      movel(pose_trans(ref_frame,p[0.017484, 0.129054, -0.000125, -0.013708, 3.141563, 0.000000]),accel_mss,speed_ms,0,0.001)
      movel(pose_trans(ref_frame,p[0.017661, 0.129058, -0.000125, -0.013708, 3.141563, -0.000000]),accel_mss,speed_ms,0,0.001)
      movel(pose_trans(ref_frame,p[0.017837, 0.129065, -0.000125, -0.013708, 3.141563, -0.000000]),accel_mss,speed_ms,0,0.001)
      movel(pose_trans(ref_frame,p[0.017988, 0.129072, -0.000125, -0.013708, 3.141563, -0.000000]),accel_mss,speed_ms,0,0.001)
      movel(pose_trans(ref_frame,p[0.018138, 0.129080, -0.000125, -0.013708, 3.141563, 0.000000]),accel_mss,speed_ms,0,0.001)
      movel(pose_trans(ref_frame,p[0.018163, 0.129086, -0.000125, -0.013708, 3.141563, 0.000000]),accel_mss,speed_ms,0,0.001)
      movel(pose_trans(ref_frame,p[0.018184, 0.129101, -0.000125, -0.013708, 3.141563, -0.000000]),accel_mss,speed_ms,0,0.001)
      movel(pose_trans(ref_frame,p[0.018198, 0.129121, -0.000125, -0.013708, 3.141563, 0.000000]),accel_mss,speed_ms,0,0.001)
      movel(pose_trans(ref_frame,p[0.018205, 0.129145, -0.000125, -0.013708, 3.141563, 0.000000]),accel_mss,speed_ms,0,0.001)
      movel(pose_trans(ref_frame,p[0.018212, 0.129253, -0.000125, -0.013708, 3.141563, -0.000000]),accel_mss,speed_ms,0,0.001)
      movel(pose_trans(ref_frame,p[0.018218, 0.129360, -0.000125, -0.013708, 3.141563, -0.000000]),accel_mss,speed_ms,0,0.001)
      movel(pose_trans(ref_frame,p[0.018224, 0.129489, -0.000125, -0.013708, 3.141563, -0.000000]),accel_mss,speed_ms,0,0.001)
      movel(pose_trans(ref_frame,p[0.018228, 0.129617, -0.000125, -0.013708, 3.141563, 0.000000]),accel_mss,speed_ms,0,0.001)
      movel(pose_trans(ref_frame,p[0.018229, 0.129765, -0.000125, -0.013708, 3.141563, 0.000000]),accel_mss,speed_ms,0,0.001)
      movel(pose_trans(ref_frame,p[0.018229, 0.129912, -0.000125, -0.013708, 3.141563, -0.000000]),accel_mss,speed_ms,0,0.001)
      movel(pose_trans(ref_frame,p[0.018230, 0.130063, -0.000125, -0.013708, 3.141563, -0.000000]),accel_mss,speed_ms,0,0.001)
      movel(pose_trans(ref_frame,p[0.018236, 0.130213, -0.000125, -0.013708, 3.141563, -0.000000]),accel_mss,speed_ms,0,0.001)
      movel(pose_trans(ref_frame,p[0.018246, 0.130351, -0.000125, -0.013708, 3.141563, -0.000000]),accel_mss,speed_ms,0,0.001)
      movel(pose_trans(ref_frame,p[0.018262, 0.130488, -0.000125, -0.013708, 3.141563, -0.000000]),accel_mss,speed_ms,0,0.001)
      movel(pose_trans(ref_frame,p[0.018280, 0.130600, -0.000125, -0.013708, 3.141563, 0.000000]),accel_mss,speed_ms,0,0.001)
      movel(pose_trans(ref_frame,p[0.018302, 0.130711, -0.000125, -0.013708, 3.141563, -0.000000]),accel_mss,speed_ms,0,0.001)
      movel(pose_trans(ref_frame,p[0.018321, 0.130761, -0.000125, -0.013708, 3.141563, 0.000000]),accel_mss,speed_ms,0,0.001)
      movel(pose_trans(ref_frame,p[0.018353, 0.130804, -0.000125, -0.013708, 3.141563, 0.000000]),accel_mss,speed_ms,0,0.001)
      movel(pose_trans(ref_frame,p[0.018453, 0.130875, -0.000125, -0.013708, 3.141563, 0.000000]),accel_mss,speed_ms,0,0.001)
      movel(pose_trans(ref_frame,p[0.018570, 0.130910, -0.000125, -0.013708, 3.141563, -0.000000]),accel_mss,speed_ms,0,0.001)
      movel(pose_trans(ref_frame,p[0.018832, 0.130940, -0.000125, -0.013708, 3.141563, -0.000000]),accel_mss,speed_ms,0,0.001)
      movel(pose_trans(ref_frame,p[0.019095, 0.130958, -0.000125, -0.013708, 3.141563, -0.000000]),accel_mss,speed_ms,0,0.001)
      movel(pose_trans(ref_frame,p[0.019359, 0.130965, -0.000125, -0.013708, 3.141563, -0.000000]),accel_mss,speed_ms,0,0.001)
      movel(pose_trans(ref_frame,p[0.019623, 0.130962, -0.000125, -0.013708, 3.141563, 0.000000]),accel_mss,speed_ms,0,0.001)
      movel(pose_trans(ref_frame,p[0.019732, 0.130938, -0.000125, -0.013708, 3.141563, -0.000000]),accel_mss,speed_ms,0,0.001)
      movel(pose_trans(ref_frame,p[0.019825, 0.130874, -0.000125, -0.013708, 3.141563, -0.000000]),accel_mss,speed_ms,0,0.001)
      movel(pose_trans(ref_frame,p[0.019913, 0.130742, -0.000125, -0.013708, 3.141563, -0.000000]),accel_mss,speed_ms,0,0.001)
      movel(pose_trans(ref_frame,p[0.019945, 0.130587, -0.000125, -0.013708, 3.141563, -0.000000]),accel_mss,speed_ms,0,0.001)
      movel(pose_trans(ref_frame,p[0.019942, 0.129872, -0.000125, -0.013708, 3.141563, -0.000000]),accel_mss,speed_ms,0,0.001)
      movel(pose_trans(ref_frame,p[0.019933, 0.129158, -0.000125, -0.013708, 3.141563, -0.000000]),accel_mss,speed_ms,0,0.001)
      movel(pose_trans(ref_frame,p[0.019916, 0.128446, -0.000125, -0.013708, 3.141563, -0.000000]),accel_mss,speed_ms,0,0.001)
      movel(pose_trans(ref_frame,p[0.019891, 0.127733, -0.000125, -0.013708, 3.141563, -0.000000]),accel_mss,speed_ms,0,0.001)
      movel(pose_trans(ref_frame,p[0.019854, 0.127574, -0.000125, -0.013708, 3.141563, 0.000000]),accel_mss,speed_ms,0,0.001)
      movel(pose_trans(ref_frame,p[0.019761, 0.127438, -0.000125, -0.013708, 3.141563, -0.000000]),accel_mss,speed_ms,0,0.001)
      movel(pose_trans(ref_frame,p[0.019695, 0.127391, -0.000125, -0.013708, 3.141563, 0.000000]),accel_mss,speed_ms,0,0.001)
      movel(pose_trans(ref_frame,p[0.019616, 0.127368, -0.000125, -0.013708, 3.141563, -0.000000]),accel_mss,speed_ms,0,0.001)
      movel(pose_trans(ref_frame,p[0.019379, 0.127340, -0.000125, -0.013708, 3.141563, 0.000000]),accel_mss,speed_ms,0,0.001)
      movel(pose_trans(ref_frame,p[0.019142, 0.127318, -0.000125, -0.013708, 3.141563, -0.000000]),accel_mss,speed_ms,0,0.001)
      movel(pose_trans(ref_frame,p[0.018838, 0.127297, -0.000125, -0.013708, 3.141563, 0.000000]),accel_mss,speed_ms,0,0.001)
      movel(pose_trans(ref_frame,p[0.018535, 0.127285, -0.000125, -0.013708, 3.141563, 0.000000]),accel_mss,speed_ms,0,0.001)
      movel(pose_trans(ref_frame,p[0.018165, 0.127278, -0.000125, -0.013708, 3.141563, -0.000000]),accel_mss,speed_ms,0,0.001)
      movel(pose_trans(ref_frame,p[0.017795, 0.127276, -0.000125, -0.013708, 3.141563, -0.000000]),accel_mss,speed_ms,0,0.001)
      movel(pose_trans(ref_frame,p[0.015998, 0.127282, -0.000125, -0.013708, 3.141563, -0.000000]),accel_mss,speed_ms,0,0.001)
      movel(pose_trans(ref_frame,p[0.016051, 0.074830, -0.000125, -0.013708, 3.141563, 0.000000]),accel_mss,speed_ms,0,0.001)
      movel(pose_trans(ref_frame,p[0.016105, 0.022378, -0.000125, -0.013708, 3.141563, -0.000000]),accel_mss,speed_ms,0,0.001)
      movel(pose_trans(ref_frame,p[0.017978, 0.022373, -0.000125, -0.013708, 3.141563, -0.000000]),accel_mss,speed_ms,0,0.001)
      movel(pose_trans(ref_frame,p[0.018340, 0.022370, -0.000125, -0.013708, 3.141563, -0.000000]),accel_mss,speed_ms,0,0.001)
      movel(pose_trans(ref_frame,p[0.018702, 0.022365, -0.000125, -0.013708, 3.141563, -0.000000]),accel_mss,speed_ms,0,0.001)
      movel(pose_trans(ref_frame,p[0.019012, 0.022358, -0.000125, -0.013708, 3.141563, -0.000000]),accel_mss,speed_ms,0,0.001)
      movel(pose_trans(ref_frame,p[0.019323, 0.022347, -0.000125, -0.013708, 3.141563, -0.000000]),accel_mss,speed_ms,0,0.001)
      movel(pose_trans(ref_frame,p[0.019591, 0.022336, -0.000125, -0.013708, 3.141563, -0.000000]),accel_mss,speed_ms,0,0.001)
      movel(pose_trans(ref_frame,p[0.019858, 0.022323, -0.000125, -0.013708, 3.141563, 0.000000]),accel_mss,speed_ms,0,0.001)
      movel(pose_trans(ref_frame,p[0.019895, 0.022315, -0.000125, -0.013708, 3.141563, -0.000000]),accel_mss,speed_ms,0,0.001)
      movel(pose_trans(ref_frame,p[0.019925, 0.022294, -0.000125, -0.013708, 3.141563, -0.000000]),accel_mss,speed_ms,0,0.001)
      movel(pose_trans(ref_frame,p[0.019999, 0.022182, -0.000125, -0.013708, 3.141563, -0.000000]),accel_mss,speed_ms,0,0.001)
      movel(pose_trans(ref_frame,p[0.020024, 0.022051, -0.000125, -0.013708, 3.141563, 0.000000]),accel_mss,speed_ms,0,0.001)
      movel(pose_trans(ref_frame,p[0.020011, 0.021314, -0.000125, -0.013708, 3.141563, -0.000000]),accel_mss,speed_ms,0,0.001)
      movel(pose_trans(ref_frame,p[0.019994, 0.020578, -0.000125, -0.013708, 3.141563, -0.000000]),accel_mss,speed_ms,0,0.001)
      movel(pose_trans(ref_frame,p[0.019971, 0.019844, -0.000125, -0.013708, 3.141563, -0.000000]),accel_mss,speed_ms,0,0.001)
      movel(pose_trans(ref_frame,p[0.019943, 0.019110, -0.000125, -0.013708, 3.141563, -0.000000]),accel_mss,speed_ms,0,0.001)
      movel(pose_trans(ref_frame,p[0.019911, 0.018972, -0.000125, -0.013708, 3.141563, -0.000000]),accel_mss,speed_ms,0,0.001)
      movel(pose_trans(ref_frame,p[0.019832, 0.018856, -0.000125, -0.013708, 3.141563, -0.000000]),accel_mss,speed_ms,0,0.001)
      movel(pose_trans(ref_frame,p[0.019724, 0.018779, -0.000125, -0.013708, 3.141563, -0.000000]),accel_mss,speed_ms,0,0.001)
      movel(pose_trans(ref_frame,p[0.019598, 0.018740, -0.000125, -0.013708, 3.141563, 0.000000]),accel_mss,speed_ms,0,0.001)
      movel(pose_trans(ref_frame,p[0.019363, 0.018715, -0.000125, -0.013708, 3.141563, -0.000000]),accel_mss,speed_ms,0,0.001)
      movel(pose_trans(ref_frame,p[0.019127, 0.018706, -0.000125, -0.013708, 3.141563, 0.000000]),accel_mss,speed_ms,0,0.001)
      movel(pose_trans(ref_frame,p[0.018891, 0.018713, -0.000125, -0.013708, 3.141563, -0.000000]),accel_mss,speed_ms,0,0.001)
      movel(pose_trans(ref_frame,p[0.018657, 0.018735, -0.000125, -0.013708, 3.141563, 0.000000]),accel_mss,speed_ms,0,0.001)
      movel(pose_trans(ref_frame,p[0.018531, 0.018772, -0.000125, -0.013708, 3.141563, 0.000000]),accel_mss,speed_ms,0,0.001)
      movel(pose_trans(ref_frame,p[0.018424, 0.018848, -0.000125, -0.013708, 3.141563, -0.000000]),accel_mss,speed_ms,0,0.001)
      movel(pose_trans(ref_frame,p[0.018391, 0.018893, -0.000125, -0.013708, 3.141563, -0.000000]),accel_mss,speed_ms,0,0.001)
      movel(pose_trans(ref_frame,p[0.018370, 0.018945, -0.000125, -0.013708, 3.141563, -0.000000]),accel_mss,speed_ms,0,0.001)
      movel(pose_trans(ref_frame,p[0.018345, 0.019059, -0.000125, -0.013708, 3.141563, -0.000000]),accel_mss,speed_ms,0,0.001)
      movel(pose_trans(ref_frame,p[0.018324, 0.019174, -0.000125, -0.013708, 3.141563, -0.000000]),accel_mss,speed_ms,0,0.001)
      movel(pose_trans(ref_frame,p[0.018304, 0.019315, -0.000125, -0.013708, 3.141563, 0.000000]),accel_mss,speed_ms,0,0.001)
      movel(pose_trans(ref_frame,p[0.018290, 0.019456, -0.000125, -0.013708, 3.141563, -0.000000]),accel_mss,speed_ms,0,0.001)
      movel(pose_trans(ref_frame,p[0.018281, 0.019610, -0.000125, -0.013708, 3.141563, -0.000000]),accel_mss,speed_ms,0,0.001)
      movel(pose_trans(ref_frame,p[0.018276, 0.019764, -0.000125, -0.013708, 3.141563, -0.000000]),accel_mss,speed_ms,0,0.001)
      movel(pose_trans(ref_frame,p[0.018273, 0.019916, -0.000125, -0.013708, 3.141563, -0.000000]),accel_mss,speed_ms,0,0.001)
      movel(pose_trans(ref_frame,p[0.018267, 0.020067, -0.000125, -0.013708, 3.141563, 0.000000]),accel_mss,speed_ms,0,0.001)
      movel(pose_trans(ref_frame,p[0.018260, 0.020200, -0.000125, -0.013708, 3.141563, -0.000000]),accel_mss,speed_ms,0,0.001)
      movel(pose_trans(ref_frame,p[0.018249, 0.020333, -0.000125, -0.013708, 3.141563, -0.000000]),accel_mss,speed_ms,0,0.001)
      movel(pose_trans(ref_frame,p[0.018239, 0.020443, -0.000125, -0.013708, 3.141563, -0.000000]),accel_mss,speed_ms,0,0.001)
      movel(pose_trans(ref_frame,p[0.018227, 0.020553, -0.000125, -0.013708, 3.141563, -0.000000]),accel_mss,speed_ms,0,0.001)
      movel(pose_trans(ref_frame,p[0.018219, 0.020582, -0.000125, -0.013708, 3.141563, -0.000000]),accel_mss,speed_ms,0,0.001)
      movel(pose_trans(ref_frame,p[0.018201, 0.020606, -0.000125, -0.013708, 3.141563, -0.000000]),accel_mss,speed_ms,0,0.001)
      movel(pose_trans(ref_frame,p[0.018176, 0.020624, -0.000125, -0.013708, 3.141563, -0.000000]),accel_mss,speed_ms,0,0.001)
      movel(pose_trans(ref_frame,p[0.018146, 0.020632, -0.000125, -0.013708, 3.141563, -0.000000]),accel_mss,speed_ms,0,0.001)
      movel(pose_trans(ref_frame,p[0.018002, 0.020641, -0.000125, -0.013708, 3.141563, -0.000000]),accel_mss,speed_ms,0,0.001)
      movel(pose_trans(ref_frame,p[0.017857, 0.020649, -0.000125, -0.013708, 3.141563, -0.000000]),accel_mss,speed_ms,0,0.001)
      movel(pose_trans(ref_frame,p[0.017685, 0.020657, -0.000125, -0.013708, 3.141563, -0.000000]),accel_mss,speed_ms,0,0.001)
      movel(pose_trans(ref_frame,p[0.017514, 0.020662, -0.000125, -0.013708, 3.141563, -0.000000]),accel_mss,speed_ms,0,0.001)
      movel(pose_trans(ref_frame,p[0.017316, 0.020664, -0.000125, -0.013708, 3.141563, -0.000000]),accel_mss,speed_ms,0,0.001)
      movel(pose_trans(ref_frame,p[0.017118, 0.020664, -0.000125, -0.013708, 3.141563, -0.000000]),accel_mss,speed_ms,0,0.001)
      movel(pose_trans(ref_frame,p[0.016098, 0.020659, -0.000125, -0.013708, 3.141563, -0.000000]),accel_mss,speed_ms,0,0.001)
      movel(pose_trans(ref_frame,p[0.016098, 0.019605, -0.000125, -0.013708, 3.141563, -0.000000]),accel_mss,speed_ms,0,0.001)
      movel(pose_trans(ref_frame,p[0.016098, 0.018551, -0.000125, -0.013708, 3.141563, 0.000000]),accel_mss,speed_ms,0,0.001)
      movel(pose_trans(ref_frame,p[0.017009, 0.018525, -0.000125, -0.013708, 3.141563, -0.000000]),accel_mss,speed_ms,0,0.001)
      movel(pose_trans(ref_frame,p[0.017185, 0.018519, -0.000125, -0.013708, 3.141563, -0.000000]),accel_mss,speed_ms,0,0.001)
      movel(pose_trans(ref_frame,p[0.017362, 0.018512, -0.000125, -0.013708, 3.141563, -0.000000]),accel_mss,speed_ms,0,0.001)
      movel(pose_trans(ref_frame,p[0.017514, 0.018504, -0.000125, -0.013708, 3.141563, -0.000000]),accel_mss,speed_ms,0,0.001)
      movel(pose_trans(ref_frame,p[0.017666, 0.018493, -0.000125, -0.013708, 3.141563, -0.000000]),accel_mss,speed_ms,0,0.001)
      movel(pose_trans(ref_frame,p[0.017796, 0.018483, -0.000125, -0.013708, 3.141563, -0.000000]),accel_mss,speed_ms,0,0.001)
      movel(pose_trans(ref_frame,p[0.017925, 0.018472, -0.000125, -0.013708, 3.141563, 0.000000]),accel_mss,speed_ms,0,0.001)
      movel(pose_trans(ref_frame,p[0.017948, 0.018466, -0.000125, -0.013708, 3.141563, 0.000000]),accel_mss,speed_ms,0,0.001)
      movel(pose_trans(ref_frame,p[0.017968, 0.018452, -0.000125, -0.013708, 3.141563, 0.000000]),accel_mss,speed_ms,0,0.001)
      movel(pose_trans(ref_frame,p[0.018022, 0.018372, -0.000125, -0.013708, 3.141563, 0.000000]),accel_mss,speed_ms,0,0.001)
      movel(pose_trans(ref_frame,p[0.018043, 0.018278, -0.000125, -0.013708, 3.141563, -0.000000]),accel_mss,speed_ms,0,0.001)
      movel(pose_trans(ref_frame,p[0.018048, 0.017994, -0.000125, -0.013708, 3.141563, -0.000000]),accel_mss,speed_ms,0,0.001)
      movel(pose_trans(ref_frame,p[0.018046, 0.017710, -0.000125, -0.013708, 3.141563, -0.000000]),accel_mss,speed_ms,0,0.001)
      movel(pose_trans(ref_frame,p[0.018037, 0.017427, -0.000125, -0.013708, 3.141563, -0.000000]),accel_mss,speed_ms,0,0.001)
      movel(pose_trans(ref_frame,p[0.018022, 0.017143, -0.000125, -0.013708, 3.141563, -0.000000]),accel_mss,speed_ms,0,0.001)
      movel(pose_trans(ref_frame,p[0.017997, 0.017047, -0.000125, -0.013708, 3.141563, -0.000000]),accel_mss,speed_ms,0,0.001)
      movel(pose_trans(ref_frame,p[0.017940, 0.016965, -0.000125, -0.013708, 3.141563, -0.000000]),accel_mss,speed_ms,0,0.001)
      movel(pose_trans(ref_frame,p[0.017895, 0.016930, -0.000125, -0.013708, 3.141563, -0.000000]),accel_mss,speed_ms,0,0.001)
      movel(pose_trans(ref_frame,p[0.017843, 0.016910, -0.000125, -0.013708, 3.141563, -0.000000]),accel_mss,speed_ms,0,0.001)
      movel(pose_trans(ref_frame,p[0.017730, 0.016885, -0.000125, -0.013708, 3.141563, -0.000000]),accel_mss,speed_ms,0,0.001)
      movel(pose_trans(ref_frame,p[0.017617, 0.016865, -0.000125, -0.013708, 3.141563, -0.000000]),accel_mss,speed_ms,0,0.001)
      movel(pose_trans(ref_frame,p[0.017478, 0.016846, -0.000125, -0.013708, 3.141563, -0.000000]),accel_mss,speed_ms,0,0.001)
      movel(pose_trans(ref_frame,p[0.017339, 0.016833, -0.000125, -0.013708, 3.141563, -0.000000]),accel_mss,speed_ms,0,0.001)
      movel(pose_trans(ref_frame,p[0.017188, 0.016825, -0.000125, -0.013708, 3.141563, -0.000000]),accel_mss,speed_ms,0,0.001)
      movel(pose_trans(ref_frame,p[0.017036, 0.016823, -0.000125, -0.013708, 3.141563, 0.000000]),accel_mss,speed_ms,0,0.001)
      movel(pose_trans(ref_frame,p[0.016887, 0.016821, -0.000125, -0.013708, 3.141563, -0.000000]),accel_mss,speed_ms,0,0.001)
      movel(pose_trans(ref_frame,p[0.016737, 0.016816, -0.000125, -0.013708, 3.141563, -0.000000]),accel_mss,speed_ms,0,0.001)
      movel(pose_trans(ref_frame,p[0.016604, 0.016808, -0.000125, -0.013708, 3.141563, -0.000000]),accel_mss,speed_ms,0,0.001)
      movel(pose_trans(ref_frame,p[0.016470, 0.016796, -0.000125, -0.013708, 3.141563, -0.000000]),accel_mss,speed_ms,0,0.001)
      movel(pose_trans(ref_frame,p[0.016361, 0.016784, -0.000125, -0.013708, 3.141563, -0.000000]),accel_mss,speed_ms,0,0.001)
      movel(pose_trans(ref_frame,p[0.016252, 0.016769, -0.000125, -0.013708, 3.141563, -0.000000]),accel_mss,speed_ms,0,0.001)
      movel(pose_trans(ref_frame,p[0.016214, 0.016758, -0.000125, -0.013708, 3.141563, -0.000000]),accel_mss,speed_ms,0,0.001)
      movel(pose_trans(ref_frame,p[0.016182, 0.016736, -0.000125, -0.013708, 3.141563, -0.000000]),accel_mss,speed_ms,0,0.001)
      movel(pose_trans(ref_frame,p[0.016158, 0.016703, -0.000125, -0.013708, 3.141563, -0.000000]),accel_mss,speed_ms,0,0.001)
      movel(pose_trans(ref_frame,p[0.016146, 0.016664, -0.000125, -0.013708, 3.141563, -0.000000]),accel_mss,speed_ms,0,0.001)
      movel(pose_trans(ref_frame,p[0.016132, 0.016520, -0.000125, -0.013708, 3.141563, -0.000000]),accel_mss,speed_ms,0,0.001)
      movel(pose_trans(ref_frame,p[0.016119, 0.016377, -0.000125, -0.013708, 3.141563, -0.000000]),accel_mss,speed_ms,0,0.001)
      movel(pose_trans(ref_frame,p[0.016108, 0.016203, -0.000125, -0.013708, 3.141563, 0.000000]),accel_mss,speed_ms,0,0.001)
      movel(pose_trans(ref_frame,p[0.016101, 0.016029, -0.000125, -0.013708, 3.141563, 0.000000]),accel_mss,speed_ms,0,0.001)
      movel(pose_trans(ref_frame,p[0.016097, 0.015831, -0.000125, -0.013708, 3.141563, -0.000000]),accel_mss,speed_ms,0,0.001)
      movel(pose_trans(ref_frame,p[0.016097, 0.015633, -0.000125, -0.013708, 3.141563, -0.000000]),accel_mss,speed_ms,0,0.001)
      movel(pose_trans(ref_frame,p[0.016102, 0.014616, -0.000125, -0.013708, 3.141563, -0.000000]),accel_mss,speed_ms,0,0.001)
      movel(pose_trans(ref_frame,p[0.016912, 0.014609, -0.000125, -0.013708, 3.141563, -0.000000]),accel_mss,speed_ms,0,0.001)
      movel(pose_trans(ref_frame,p[0.017074, 0.014605, -0.000125, -0.013708, 3.141563, -0.000000]),accel_mss,speed_ms,0,0.001)
      movel(pose_trans(ref_frame,p[0.017235, 0.014595, -0.000125, -0.013708, 3.141563, -0.000000]),accel_mss,speed_ms,0,0.001)
      movel(pose_trans(ref_frame,p[0.017384, 0.014579, -0.000125, -0.013708, 3.141563, -0.000000]),accel_mss,speed_ms,0,0.001)
      movel(pose_trans(ref_frame,p[0.017533, 0.014557, -0.000125, -0.013708, 3.141563, -0.000000]),accel_mss,speed_ms,0,0.001)
      movel(pose_trans(ref_frame,p[0.017655, 0.014533, -0.000125, -0.013708, 3.141563, -0.000000]),accel_mss,speed_ms,0,0.001)
      movel(pose_trans(ref_frame,p[0.017776, 0.014503, -0.000125, -0.013708, 3.141563, -0.000000]),accel_mss,speed_ms,0,0.001)
      movel(pose_trans(ref_frame,p[0.017836, 0.014478, -0.000125, -0.013708, 3.141563, -0.000000]),accel_mss,speed_ms,0,0.001)
      movel(pose_trans(ref_frame,p[0.017888, 0.014438, -0.000125, -0.013708, 3.141563, -0.000000]),accel_mss,speed_ms,0,0.001)
      movel(pose_trans(ref_frame,p[0.017927, 0.014387, -0.000125, -0.013708, 3.141563, -0.000000]),accel_mss,speed_ms,0,0.001)
      movel(pose_trans(ref_frame,p[0.017952, 0.014327, -0.000125, -0.013708, 3.141563, -0.000000]),accel_mss,speed_ms,0,0.001)
      movel(pose_trans(ref_frame,p[0.017982, 0.014206, -0.000125, -0.013708, 3.141563, -0.000000]),accel_mss,speed_ms,0,0.001)
      movel(pose_trans(ref_frame,p[0.018006, 0.014084, -0.000125, -0.013708, 3.141563, 0.000000]),accel_mss,speed_ms,0,0.001)
      movel(pose_trans(ref_frame,p[0.018028, 0.013935, -0.000125, -0.013708, 3.141563, 0.000000]),accel_mss,speed_ms,0,0.001)
      movel(pose_trans(ref_frame,p[0.018044, 0.013786, -0.000125, -0.013708, 3.141563, -0.000000]),accel_mss,speed_ms,0,0.001)
      movel(pose_trans(ref_frame,p[0.018054, 0.013625, -0.000125, -0.013708, 3.141563, -0.000000]),accel_mss,speed_ms,0,0.001)
      movel(pose_trans(ref_frame,p[0.018058, 0.013463, -0.000125, -0.013708, 3.141563, -0.000000]),accel_mss,speed_ms,0,0.001)
      movel(pose_trans(ref_frame,p[0.018065, 0.012653, -0.000125, -0.013708, 3.141563, -0.000000]),accel_mss,speed_ms,0,0.001)
      movel(pose_trans(ref_frame,p[0.019082, 0.012648, -0.000125, -0.013708, 3.141563, -0.000000]),accel_mss,speed_ms,0,0.001)
      movel(pose_trans(ref_frame,p[0.019281, 0.012648, -0.000125, -0.013708, 3.141563, 0.000000]),accel_mss,speed_ms,0,0.001)
      movel(pose_trans(ref_frame,p[0.019479, 0.012653, -0.000125, -0.013708, 3.141563, -0.000000]),accel_mss,speed_ms,0,0.001)
      movel(pose_trans(ref_frame,p[0.019654, 0.012660, -0.000125, -0.013708, 3.141563, -0.000000]),accel_mss,speed_ms,0,0.001)
      movel(pose_trans(ref_frame,p[0.019830, 0.012673, -0.000125, -0.013708, 3.141563, -0.000000]),accel_mss,speed_ms,0,0.001)
      movel(pose_trans(ref_frame,p[0.019974, 0.012686, -0.000125, -0.013708, 3.141563, -0.000000]),accel_mss,speed_ms,0,0.001)
      movel(pose_trans(ref_frame,p[0.020118, 0.012702, -0.000125, -0.013708, 3.141563, -0.000000]),accel_mss,speed_ms,0,0.001)
      movel(pose_trans(ref_frame,p[0.020161, 0.012715, -0.000125, -0.013708, 3.141563, -0.000000]),accel_mss,speed_ms,0,0.001)
      movel(pose_trans(ref_frame,p[0.020198, 0.012741, -0.000125, -0.013708, 3.141563, -0.000000]),accel_mss,speed_ms,0,0.001)
      movel(pose_trans(ref_frame,p[0.020223, 0.012775, -0.000125, -0.013708, 3.141563, -0.000000]),accel_mss,speed_ms,0,0.001)
      movel(pose_trans(ref_frame,p[0.020235, 0.012815, -0.000125, -0.013708, 3.141563, -0.000000]),accel_mss,speed_ms,0,0.001)
      movel(pose_trans(ref_frame,p[0.020248, 0.012921, -0.000125, -0.013708, 3.141563, -0.000000]),accel_mss,speed_ms,0,0.001)
      movel(pose_trans(ref_frame,p[0.020259, 0.013027, -0.000125, -0.013708, 3.141563, -0.000000]),accel_mss,speed_ms,0,0.001)
      movel(pose_trans(ref_frame,p[0.020267, 0.013157, -0.000125, -0.013708, 3.141563, -0.000000]),accel_mss,speed_ms,0,0.001)
      movel(pose_trans(ref_frame,p[0.020271, 0.013287, -0.000125, -0.013708, 3.141563, -0.000000]),accel_mss,speed_ms,0,0.001)
      movel(pose_trans(ref_frame,p[0.020270, 0.013432, -0.000125, -0.013708, 3.141563, 0.000000]),accel_mss,speed_ms,0,0.001)
      movel(pose_trans(ref_frame,p[0.020266, 0.013577, -0.000125, -0.013708, 3.141563, 0.000000]),accel_mss,speed_ms,0,0.001)
      movel(pose_trans(ref_frame,p[0.020263, 0.013723, -0.000125, -0.013708, 3.141563, -0.000000]),accel_mss,speed_ms,0,0.001)
      movel(pose_trans(ref_frame,p[0.020266, 0.013870, -0.000125, -0.013708, 3.141563, -0.000000]),accel_mss,speed_ms,0,0.001)
      movel(pose_trans(ref_frame,p[0.020275, 0.014006, -0.000125, -0.013708, 3.141563, -0.000000]),accel_mss,speed_ms,0,0.001)
      movel(pose_trans(ref_frame,p[0.020290, 0.014142, -0.000125, -0.013708, 3.141563, 0.000000]),accel_mss,speed_ms,0,0.001)
      movel(pose_trans(ref_frame,p[0.020308, 0.014253, -0.000125, -0.013708, 3.141563, -0.000000]),accel_mss,speed_ms,0,0.001)
      movel(pose_trans(ref_frame,p[0.020331, 0.014364, -0.000125, -0.013708, 3.141563, -0.000000]),accel_mss,speed_ms,0,0.001)
      movel(pose_trans(ref_frame,p[0.020353, 0.014419, -0.000125, -0.013708, 3.141563, -0.000000]),accel_mss,speed_ms,0,0.001)
      movel(pose_trans(ref_frame,p[0.020389, 0.014466, -0.000125, -0.013708, 3.141563, -0.000000]),accel_mss,speed_ms,0,0.001)
      movel(pose_trans(ref_frame,p[0.020498, 0.014544, -0.000125, -0.013708, 3.141563, -0.000000]),accel_mss,speed_ms,0,0.001)
      movel(pose_trans(ref_frame,p[0.020626, 0.014582, -0.000125, -0.013708, 3.141563, -0.000000]),accel_mss,speed_ms,0,0.001)
      movel(pose_trans(ref_frame,p[0.020861, 0.014602, -0.000125, -0.013708, 3.141563, -0.000000]),accel_mss,speed_ms,0,0.001)
      movel(pose_trans(ref_frame,p[0.021097, 0.014605, -0.000125, -0.013708, 3.141563, -0.000000]),accel_mss,speed_ms,0,0.001)
      movel(pose_trans(ref_frame,p[0.021333, 0.014592, -0.000125, -0.013708, 3.141563, -0.000000]),accel_mss,speed_ms,0,0.001)
      movel(pose_trans(ref_frame,p[0.021568, 0.014562, -0.000125, -0.013708, 3.141563, -0.000000]),accel_mss,speed_ms,0,0.001)
      movel(pose_trans(ref_frame,p[0.021700, 0.014519, -0.000125, -0.013708, 3.141563, -0.000000]),accel_mss,speed_ms,0,0.001)
      movel(pose_trans(ref_frame,p[0.021812, 0.014437, -0.000125, -0.013708, 3.141563, -0.000000]),accel_mss,speed_ms,0,0.001)
      movel(pose_trans(ref_frame,p[0.021851, 0.014386, -0.000125, -0.013708, 3.141563, -0.000000]),accel_mss,speed_ms,0,0.001)
      movel(pose_trans(ref_frame,p[0.021876, 0.014326, -0.000125, -0.013708, 3.141563, -0.000000]),accel_mss,speed_ms,0,0.001)
      movel(pose_trans(ref_frame,p[0.021905, 0.014205, -0.000125, -0.013708, 3.141563, 0.000000]),accel_mss,speed_ms,0,0.001)
      movel(pose_trans(ref_frame,p[0.021929, 0.014083, -0.000125, -0.013708, 3.141563, -0.000000]),accel_mss,speed_ms,0,0.001)
      movel(pose_trans(ref_frame,p[0.021951, 0.013934, -0.000125, -0.013708, 3.141563, -0.000000]),accel_mss,speed_ms,0,0.001)
      movel(pose_trans(ref_frame,p[0.021967, 0.013784, -0.000125, -0.013708, 3.141563, -0.000000]),accel_mss,speed_ms,0,0.001)
      movel(pose_trans(ref_frame,p[0.021977, 0.013623, -0.000125, -0.013708, 3.141563, -0.000000]),accel_mss,speed_ms,0,0.001)
      movel(pose_trans(ref_frame,p[0.021982, 0.013462, -0.000125, -0.013708, 3.141563, 0.000000]),accel_mss,speed_ms,0,0.001)
      movel(pose_trans(ref_frame,p[0.021988, 0.012649, -0.000125, -0.013708, 3.141563, -0.000000]),accel_mss,speed_ms,0,0.001)
      movel(pose_trans(ref_frame,p[0.023048, 0.012649, -0.000125, -0.013708, 3.141563, -0.000000]),accel_mss,speed_ms,0,0.001)
      movel(pose_trans(ref_frame,p[0.024108, 0.012649, -0.000125, -0.013708, 3.141563, -0.000000]),accel_mss,speed_ms,0,0.001)
      movel(pose_trans(ref_frame,p[0.024113, 0.013669, -0.000125, -0.013708, 3.141563, -0.000000]),accel_mss,speed_ms,0,0.001)
      movel(pose_trans(ref_frame,p[0.024113, 0.013866, -0.000125, -0.013708, 3.141563, -0.000000]),accel_mss,speed_ms,0,0.001)
      movel(pose_trans(ref_frame,p[0.024112, 0.014063, -0.000125, -0.013708, 3.141563, -0.000000]),accel_mss,speed_ms,0,0.001)
      movel(pose_trans(ref_frame,p[0.024109, 0.014233, -0.000125, -0.013708, 3.141563, 0.000000]),accel_mss,speed_ms,0,0.001)
      movel(pose_trans(ref_frame,p[0.024103, 0.014403, -0.000125, -0.013708, 3.141563, -0.000000]),accel_mss,speed_ms,0,0.001)
      movel(pose_trans(ref_frame,p[0.024098, 0.014548, -0.000125, -0.013708, 3.141563, -0.000000]),accel_mss,speed_ms,0,0.001)
      movel(pose_trans(ref_frame,p[0.024091, 0.014693, -0.000125, -0.013708, 3.141563, -0.000000]),accel_mss,speed_ms,0,0.001)
      movel(pose_trans(ref_frame,p[0.024086, 0.014716, -0.000125, -0.013708, 3.141563, -0.000000]),accel_mss,speed_ms,0,0.001)
      movel(pose_trans(ref_frame,p[0.024073, 0.014735, -0.000125, -0.013708, 3.141563, -0.000000]),accel_mss,speed_ms,0,0.001)
      movel(pose_trans(ref_frame,p[0.024054, 0.014748, -0.000125, -0.013708, 3.141563, -0.000000]),accel_mss,speed_ms,0,0.001)
      movel(pose_trans(ref_frame,p[0.024032, 0.014755, -0.000125, -0.013708, 3.141563, -0.000000]),accel_mss,speed_ms,0,0.001)
      movel(pose_trans(ref_frame,p[0.023918, 0.014768, -0.000125, -0.013708, 3.141563, -0.000000]),accel_mss,speed_ms,0,0.001)
      movel(pose_trans(ref_frame,p[0.023803, 0.014780, -0.000125, -0.013708, 3.141563, -0.000000]),accel_mss,speed_ms,0,0.001)
      movel(pose_trans(ref_frame,p[0.023667, 0.014793, -0.000125, -0.013708, 3.141563, -0.000000]),accel_mss,speed_ms,0,0.001)
      movel(pose_trans(ref_frame,p[0.023532, 0.014804, -0.000125, -0.013708, 3.141563, 0.000000]),accel_mss,speed_ms,0,0.001)
      movel(pose_trans(ref_frame,p[0.023375, 0.014815, -0.000125, -0.013708, 3.141563, 0.000000]),accel_mss,speed_ms,0,0.001)
      movel(pose_trans(ref_frame,p[0.023218, 0.014824, -0.000125, -0.013708, 3.141563, -0.000000]),accel_mss,speed_ms,0,0.001)
      movel(pose_trans(ref_frame,p[0.023059, 0.014835, -0.000125, -0.013708, 3.141563, -0.000000]),accel_mss,speed_ms,0,0.001)
      movel(pose_trans(ref_frame,p[0.022899, 0.014850, -0.000125, -0.013708, 3.141563, 0.000000]),accel_mss,speed_ms,0,0.001)
      movel(pose_trans(ref_frame,p[0.022753, 0.014869, -0.000125, -0.013708, 3.141563, -0.000000]),accel_mss,speed_ms,0,0.001)
      movel(pose_trans(ref_frame,p[0.022608, 0.014893, -0.000125, -0.013708, 3.141563, -0.000000]),accel_mss,speed_ms,0,0.001)
      movel(pose_trans(ref_frame,p[0.022490, 0.014917, -0.000125, -0.013708, 3.141563, -0.000000]),accel_mss,speed_ms,0,0.001)
      movel(pose_trans(ref_frame,p[0.022372, 0.014945, -0.000125, -0.013708, 3.141563, -0.000000]),accel_mss,speed_ms,0,0.001)
      movel(pose_trans(ref_frame,p[0.022321, 0.014966, -0.000125, -0.013708, 3.141563, -0.000000]),accel_mss,speed_ms,0,0.001)
      movel(pose_trans(ref_frame,p[0.022276, 0.014999, -0.000125, -0.013708, 3.141563, -0.000000]),accel_mss,speed_ms,0,0.001)
      movel(pose_trans(ref_frame,p[0.022205, 0.015098, -0.000125, -0.013708, 3.141563, 0.000000]),accel_mss,speed_ms,0,0.001)
      movel(pose_trans(ref_frame,p[0.022173, 0.015216, -0.000125, -0.013708, 3.141563, -0.000000]),accel_mss,speed_ms,0,0.001)
      movel(pose_trans(ref_frame,p[0.022157, 0.015451, -0.000125, -0.013708, 3.141563, -0.000000]),accel_mss,speed_ms,0,0.001)
      movel(pose_trans(ref_frame,p[0.022155, 0.015687, -0.000125, -0.013708, 3.141563, -0.000000]),accel_mss,speed_ms,0,0.001)
      movel(pose_trans(ref_frame,p[0.022167, 0.015923, -0.000125, -0.013708, 3.141563, -0.000000]),accel_mss,speed_ms,0,0.001)
      movel(pose_trans(ref_frame,p[0.022193, 0.016158, -0.000125, -0.013708, 3.141563, 0.000000]),accel_mss,speed_ms,0,0.001)
      movel(pose_trans(ref_frame,p[0.022232, 0.016280, -0.000125, -0.013708, 3.141563, -0.000000]),accel_mss,speed_ms,0,0.001)
      movel(pose_trans(ref_frame,p[0.022306, 0.016384, -0.000125, -0.013708, 3.141563, -0.000000]),accel_mss,speed_ms,0,0.001)
      movel(pose_trans(ref_frame,p[0.022407, 0.016453, -0.000125, -0.013708, 3.141563, -0.000000]),accel_mss,speed_ms,0,0.001)
      movel(pose_trans(ref_frame,p[0.022526, 0.016479, -0.000125, -0.013708, 3.141563, -0.000000]),accel_mss,speed_ms,0,0.001)
      movel(pose_trans(ref_frame,p[0.023281, 0.016501, -0.000125, -0.013708, 3.141563, -0.000000]),accel_mss,speed_ms,0,0.001)
      movel(pose_trans(ref_frame,p[0.024036, 0.016519, -0.000125, -0.013708, 3.141563, -0.000000]),accel_mss,speed_ms,0,0.001)
      movel(pose_trans(ref_frame,p[0.024793, 0.016533, -0.000125, -0.013708, 3.141563, -0.000000]),accel_mss,speed_ms,0,0.001)
      movel(pose_trans(ref_frame,p[0.025550, 0.016544, -0.000125, -0.013708, 3.141563, 0.000000]),accel_mss,speed_ms,0,0.001)
      movel(pose_trans(ref_frame,p[0.025665, 0.016522, -0.000125, -0.013708, 3.141563, 0.000000]),accel_mss,speed_ms,0,0.001)
      movel(pose_trans(ref_frame,p[0.025762, 0.016457, -0.000125, -0.013708, 3.141563, -0.000000]),accel_mss,speed_ms,0,0.001)
      movel(pose_trans(ref_frame,p[0.025778, 0.016434, -0.000125, -0.013708, 3.141563, -0.000000]),accel_mss,speed_ms,0,0.001)
      movel(pose_trans(ref_frame,p[0.025784, 0.016406, -0.000125, -0.013708, 3.141563, -0.000000]),accel_mss,speed_ms,0,0.001)
      movel(pose_trans(ref_frame,p[0.025793, 0.016137, -0.000125, -0.013708, 3.141563, -0.000000]),accel_mss,speed_ms,0,0.001)
      movel(pose_trans(ref_frame,p[0.025801, 0.015868, -0.000125, -0.013708, 3.141563, -0.000000]),accel_mss,speed_ms,0,0.001)
      movel(pose_trans(ref_frame,p[0.025809, 0.015559, -0.000125, -0.013708, 3.141563, 0.000000]),accel_mss,speed_ms,0,0.001)
      movel(pose_trans(ref_frame,p[0.025814, 0.015250, -0.000125, -0.013708, 3.141563, -0.000000]),accel_mss,speed_ms,0,0.001)
      movel(pose_trans(ref_frame,p[0.025818, 0.014889, -0.000125, -0.013708, 3.141563, 0.000000]),accel_mss,speed_ms,0,0.001)
      movel(pose_trans(ref_frame,p[0.025820, 0.014527, -0.000125, -0.013708, 3.141563, -0.000000]),accel_mss,speed_ms,0,0.001)
      movel(pose_trans(ref_frame,p[0.025823, 0.012652, -0.000125, -0.013708, 3.141563, 0.000000]),accel_mss,speed_ms,0,0.001)
      movel(pose_trans(ref_frame,p[0.078266, 0.012593, -0.000125, -0.013708, 3.141563, -0.000000]),accel_mss,speed_ms,0,0.001)
      movel(pose_trans(ref_frame,p[0.130708, 0.012535, -0.000125, -0.013708, 3.141563, 0.000000]),accel_mss,speed_ms,0,0.001)
      movel(pose_trans(ref_frame,p[0.130721, 0.014348, -0.000125, -0.013708, 3.141563, -0.000000]),accel_mss,speed_ms,0,0.001)
      movel(pose_trans(ref_frame,p[0.130726, 0.014701, -0.000125, -0.013708, 3.141563, -0.000000]),accel_mss,speed_ms,0,0.001)
      movel(pose_trans(ref_frame,p[0.130736, 0.015053, -0.000125, -0.013708, 3.141563, -0.000000]),accel_mss,speed_ms,0,0.001)
      movel(pose_trans(ref_frame,p[0.130750, 0.015361, -0.000125, -0.013708, 3.141563, -0.000000]),accel_mss,speed_ms,0,0.001)
      movel(pose_trans(ref_frame,p[0.130771, 0.015669, -0.000125, -0.013708, 3.141563, -0.000000]),accel_mss,speed_ms,0,0.001)
      movel(pose_trans(ref_frame,p[0.130792, 0.015926, -0.000125, -0.013708, 3.141563, 0.000000]),accel_mss,speed_ms,0,0.001)
      movel(pose_trans(ref_frame,p[0.130816, 0.016182, -0.000125, -0.013708, 3.141563, -0.000000]),accel_mss,speed_ms,0,0.001)
      movel(pose_trans(ref_frame,p[0.130834, 0.016245, -0.000125, -0.013708, 3.141563, -0.000000]),accel_mss,speed_ms,0,0.001)
      movel(pose_trans(ref_frame,p[0.130871, 0.016298, -0.000125, -0.013708, 3.141563, -0.000000]),accel_mss,speed_ms,0,0.001)
      movel(pose_trans(ref_frame,p[0.130924, 0.016335, -0.000125, -0.013708, 3.141563, -0.000000]),accel_mss,speed_ms,0,0.001)
      movel(pose_trans(ref_frame,p[0.130985, 0.016353, -0.000125, -0.013708, 3.141563, 0.000000]),accel_mss,speed_ms,0,0.001)
      movel(pose_trans(ref_frame,p[0.131215, 0.016377, -0.000125, -0.013708, 3.141563, -0.000000]),accel_mss,speed_ms,0,0.001)
      movel(pose_trans(ref_frame,p[0.131445, 0.016399, -0.000125, -0.013708, 3.141563, 0.000000]),accel_mss,speed_ms,0,0.001)
      movel(pose_trans(ref_frame,p[0.131723, 0.016419, -0.000125, -0.013708, 3.141563, 0.000000]),accel_mss,speed_ms,0,0.001)
      movel(pose_trans(ref_frame,p[0.132001, 0.016434, -0.000125, -0.013708, 3.141563, 0.000000]),accel_mss,speed_ms,0,0.001)
      movel(pose_trans(ref_frame,p[0.132317, 0.016444, -0.000125, -0.013708, 3.141563, 0.000000]),accel_mss,speed_ms,0,0.001)
      movel(pose_trans(ref_frame,p[0.132633, 0.016449, -0.000125, -0.013708, 3.141563, -0.000000]),accel_mss,speed_ms,0,0.001)
      movel(pose_trans(ref_frame,p[0.133218, 0.016450, -0.000125, -0.013708, 3.141563, -0.000000]),accel_mss,speed_ms,0,0.001)
      movel(pose_trans(ref_frame,p[0.133803, 0.016442, -0.000125, -0.013708, 3.141563, -0.000000]),accel_mss,speed_ms,0,0.001)
      movel(pose_trans(ref_frame,p[0.134003, 0.016415, -0.000125, -0.013708, 3.141563, 0.000000]),accel_mss,speed_ms,0,0.001)
      movel(pose_trans(ref_frame,p[0.134192, 0.016343, -0.000125, -0.013708, 3.141563, -0.000000]),accel_mss,speed_ms,0,0.001)
      movel(pose_trans(ref_frame,p[0.134310, 0.016242, -0.000125, -0.013708, 3.141563, 0.000000]),accel_mss,speed_ms,0,0.001)
      movel(pose_trans(ref_frame,p[0.134370, 0.016099, -0.000125, -0.013708, 3.141563, -0.000000]),accel_mss,speed_ms,0,0.001)
      movel(pose_trans(ref_frame,p[0.134407, 0.015813, -0.000125, -0.013708, 3.141563, -0.000000]),accel_mss,speed_ms,0,0.001)
      movel(pose_trans(ref_frame,p[0.134420, 0.015525, -0.000125, -0.013708, 3.141563, -0.000000]),accel_mss,speed_ms,0,0.001)
      movel(pose_trans(ref_frame,p[0.134410, 0.015304, -0.000125, -0.013708, 3.141563, -0.000000]),accel_mss,speed_ms,0,0.001)
      movel(pose_trans(ref_frame,p[0.134382, 0.015084, -0.000125, -0.013708, 3.141563, -0.000000]),accel_mss,speed_ms,0,0.001)
      movel(pose_trans(ref_frame,p[0.134337, 0.014963, -0.000125, -0.013708, 3.141563, -0.000000]),accel_mss,speed_ms,0,0.001)
      movel(pose_trans(ref_frame,p[0.134251, 0.014867, -0.000125, -0.013708, 3.141563, -0.000000]),accel_mss,speed_ms,0,0.001)
      movel(pose_trans(ref_frame,p[0.134123, 0.014796, -0.000125, -0.013708, 3.141563, -0.000000]),accel_mss,speed_ms,0,0.001)
      movel(pose_trans(ref_frame,p[0.133980, 0.014763, -0.000125, -0.013708, 3.141563, 0.000000]),accel_mss,speed_ms,0,0.001)
      movel(pose_trans(ref_frame,p[0.133681, 0.014744, -0.000125, -0.013708, 3.141563, -0.000000]),accel_mss,speed_ms,0,0.001)
      movel(pose_trans(ref_frame,p[0.133382, 0.014737, -0.000125, -0.013708, 3.141563, -0.000000]),accel_mss,speed_ms,0,0.001)
      movel(pose_trans(ref_frame,p[0.132513, 0.014735, -0.000125, -0.013708, 3.141563, -0.000000]),accel_mss,speed_ms,0,0.001)
      movel(pose_trans(ref_frame,p[0.132508, 0.013651, -0.000125, -0.013708, 3.141563, 0.000000]),accel_mss,speed_ms,0,0.001)
      movel(pose_trans(ref_frame,p[0.132503, 0.012567, -0.000125, -0.013708, 3.141563, -0.000000]),accel_mss,speed_ms,0,0.001)
      movel(pose_trans(ref_frame,p[0.133569, 0.012562, -0.000125, -0.013708, 3.141563, -0.000000]),accel_mss,speed_ms,0,0.001)
      movel(pose_trans(ref_frame,p[0.134635, 0.012557, -0.000125, -0.013708, 3.141563, -0.000000]),accel_mss,speed_ms,0,0.001)
      movel(pose_trans(ref_frame,p[0.134640, 0.013415, -0.000125, -0.013708, 3.141563, -0.000000]),accel_mss,speed_ms,0,0.001)
      movel(pose_trans(ref_frame,p[0.134644, 0.013585, -0.000125, -0.013708, 3.141563, 0.000000]),accel_mss,speed_ms,0,0.001)
      movel(pose_trans(ref_frame,p[0.134652, 0.013754, -0.000125, -0.013708, 3.141563, -0.000000]),accel_mss,speed_ms,0,0.001)
      movel(pose_trans(ref_frame,p[0.134664, 0.013907, -0.000125, -0.013708, 3.141563, 0.000000]),accel_mss,speed_ms,0,0.001)
      movel(pose_trans(ref_frame,p[0.134682, 0.014060, -0.000125, -0.013708, 3.141563, -0.000000]),accel_mss,speed_ms,0,0.001)
      movel(pose_trans(ref_frame,p[0.134702, 0.014184, -0.000125, -0.013708, 3.141563, -0.000000]),accel_mss,speed_ms,0,0.001)
      movel(pose_trans(ref_frame,p[0.134725, 0.014308, -0.000125, -0.013708, 3.141563, -0.000000]),accel_mss,speed_ms,0,0.001)
      movel(pose_trans(ref_frame,p[0.134743, 0.014360, -0.000125, -0.013708, 3.141563, -0.000000]),accel_mss,speed_ms,0,0.001)
      movel(pose_trans(ref_frame,p[0.134776, 0.014404, -0.000125, -0.013708, 3.141563, -0.000000]),accel_mss,speed_ms,0,0.001)
      movel(pose_trans(ref_frame,p[0.134843, 0.014453, -0.000125, -0.013708, 3.141563, -0.000000]),accel_mss,speed_ms,0,0.001)
      movel(pose_trans(ref_frame,p[0.134922, 0.014478, -0.000125, -0.013708, 3.141563, -0.000000]),accel_mss,speed_ms,0,0.001)
      movel(pose_trans(ref_frame,p[0.135070, 0.014497, -0.000125, -0.013708, 3.141563, -0.000000]),accel_mss,speed_ms,0,0.001)
      movel(pose_trans(ref_frame,p[0.135220, 0.014508, -0.000125, -0.013708, 3.141563, -0.000000]),accel_mss,speed_ms,0,0.001)
      movel(pose_trans(ref_frame,p[0.135415, 0.014510, -0.000125, -0.013708, 3.141563, 0.000000]),accel_mss,speed_ms,0,0.001)
      movel(pose_trans(ref_frame,p[0.135609, 0.014501, -0.000125, -0.013708, 3.141563, -0.000000]),accel_mss,speed_ms,0,0.001)
      movel(pose_trans(ref_frame,p[0.135840, 0.014481, -0.000125, -0.013708, 3.141563, 0.000000]),accel_mss,speed_ms,0,0.001)
      movel(pose_trans(ref_frame,p[0.136070, 0.014453, -0.000125, -0.013708, 3.141563, -0.000000]),accel_mss,speed_ms,0,0.001)
      movel(pose_trans(ref_frame,p[0.136146, 0.014432, -0.000125, -0.013708, 3.141563, 0.000000]),accel_mss,speed_ms,0,0.001)
      movel(pose_trans(ref_frame,p[0.136214, 0.014392, -0.000125, -0.013708, 3.141563, -0.000000]),accel_mss,speed_ms,0,0.001)
      movel(pose_trans(ref_frame,p[0.136265, 0.014337, -0.000125, -0.013708, 3.141563, -0.000000]),accel_mss,speed_ms,0,0.001)
      movel(pose_trans(ref_frame,p[0.136297, 0.014270, -0.000125, -0.013708, 3.141563, -0.000000]),accel_mss,speed_ms,0,0.001)
      movel(pose_trans(ref_frame,p[0.136323, 0.014151, -0.000125, -0.013708, 3.141563, -0.000000]),accel_mss,speed_ms,0,0.001)
      movel(pose_trans(ref_frame,p[0.136335, 0.014030, -0.000125, -0.013708, 3.141563, -0.000000]),accel_mss,speed_ms,0,0.001)
      movel(pose_trans(ref_frame,p[0.136342, 0.013761, -0.000125, -0.013708, 3.141563, -0.000000]),accel_mss,speed_ms,0,0.001)
      movel(pose_trans(ref_frame,p[0.136346, 0.013492, -0.000125, -0.013708, 3.141563, -0.000000]),accel_mss,speed_ms,0,0.001)
      movel(pose_trans(ref_frame,p[0.136352, 0.012568, -0.000125, -0.013708, 3.141563, -0.000000]),accel_mss,speed_ms,0,0.001)
      movel(pose_trans(ref_frame,p[0.137370, 0.012562, -0.000125, -0.013708, 3.141563, -0.000000]),accel_mss,speed_ms,0,0.001)
      movel(pose_trans(ref_frame,p[0.137568, 0.012563, -0.000125, -0.013708, 3.141563, -0.000000]),accel_mss,speed_ms,0,0.001)
      movel(pose_trans(ref_frame,p[0.137766, 0.012566, -0.000125, -0.013708, 3.141563, -0.000000]),accel_mss,speed_ms,0,0.001)
      movel(pose_trans(ref_frame,p[0.137940, 0.012573, -0.000125, -0.013708, 3.141563, -0.000000]),accel_mss,speed_ms,0,0.001)
      movel(pose_trans(ref_frame,p[0.138113, 0.012584, -0.000125, -0.013708, 3.141563, -0.000000]),accel_mss,speed_ms,0,0.001)
      movel(pose_trans(ref_frame,p[0.138258, 0.012595, -0.000125, -0.013708, 3.141563, -0.000000]),accel_mss,speed_ms,0,0.001)
      movel(pose_trans(ref_frame,p[0.138402, 0.012608, -0.000125, -0.013708, 3.141563, 0.000000]),accel_mss,speed_ms,0,0.001)
      movel(pose_trans(ref_frame,p[0.138440, 0.012619, -0.000125, -0.013708, 3.141563, 0.000000]),accel_mss,speed_ms,0,0.001)
      movel(pose_trans(ref_frame,p[0.138472, 0.012642, -0.000125, -0.013708, 3.141563, -0.000000]),accel_mss,speed_ms,0,0.001)
      movel(pose_trans(ref_frame,p[0.138495, 0.012673, -0.000125, -0.013708, 3.141563, -0.000000]),accel_mss,speed_ms,0,0.001)
      movel(pose_trans(ref_frame,p[0.138506, 0.012710, -0.000125, -0.013708, 3.141563, 0.000000]),accel_mss,speed_ms,0,0.001)
      movel(pose_trans(ref_frame,p[0.138521, 0.012822, -0.000125, -0.013708, 3.141563, -0.000000]),accel_mss,speed_ms,0,0.001)
      movel(pose_trans(ref_frame,p[0.138534, 0.012934, -0.000125, -0.013708, 3.141563, -0.000000]),accel_mss,speed_ms,0,0.001)
      movel(pose_trans(ref_frame,p[0.138546, 0.013072, -0.000125, -0.013708, 3.141563, -0.000000]),accel_mss,speed_ms,0,0.001)
      movel(pose_trans(ref_frame,p[0.138555, 0.013209, -0.000125, -0.013708, 3.141563, -0.000000]),accel_mss,speed_ms,0,0.001)
      movel(pose_trans(ref_frame,p[0.138561, 0.013364, -0.000125, -0.013708, 3.141563, -0.000000]),accel_mss,speed_ms,0,0.001)
      movel(pose_trans(ref_frame,p[0.138563, 0.013518, -0.000125, -0.013708, 3.141563, -0.000000]),accel_mss,speed_ms,0,0.001)
      movel(pose_trans(ref_frame,p[0.138576, 0.013815, -0.000125, -0.013708, 3.141563, -0.000000]),accel_mss,speed_ms,0,0.001)
      movel(pose_trans(ref_frame,p[0.138609, 0.014110, -0.000125, -0.013708, 3.141563, -0.000000]),accel_mss,speed_ms,0,0.001)
      movel(pose_trans(ref_frame,p[0.138661, 0.014262, -0.000125, -0.013708, 3.141563, -0.000000]),accel_mss,speed_ms,0,0.001)
      movel(pose_trans(ref_frame,p[0.138764, 0.014386, -0.000125, -0.013708, 3.141563, -0.000000]),accel_mss,speed_ms,0,0.001)
      movel(pose_trans(ref_frame,p[0.138912, 0.014473, -0.000125, -0.013708, 3.141563, 0.000000]),accel_mss,speed_ms,0,0.001)
      movel(pose_trans(ref_frame,p[0.139080, 0.014509, -0.000125, -0.013708, 3.141563, -0.000000]),accel_mss,speed_ms,0,0.001)
      movel(pose_trans(ref_frame,p[0.139426, 0.014520, -0.000125, -0.013708, 3.141563, -0.000000]),accel_mss,speed_ms,0,0.001)
      movel(pose_trans(ref_frame,p[0.139772, 0.014514, -0.000125, -0.013708, 3.141563, -0.000000]),accel_mss,speed_ms,0,0.001)
      movel(pose_trans(ref_frame,p[0.140520, 0.014483, -0.000125, -0.013708, 3.141563, -0.000000]),accel_mss,speed_ms,0,0.001)
      movel(pose_trans(ref_frame,p[0.140525, 0.015567, -0.000125, -0.013708, 3.141563, -0.000000]),accel_mss,speed_ms,0,0.001)
      movel(pose_trans(ref_frame,p[0.140530, 0.016651, -0.000125, -0.013708, 3.141563, 0.000000]),accel_mss,speed_ms,0,0.001)
      movel(pose_trans(ref_frame,p[0.139672, 0.016656, -0.000125, -0.013708, 3.141563, -0.000000]),accel_mss,speed_ms,0,0.001)
      movel(pose_trans(ref_frame,p[0.139503, 0.016659, -0.000125, -0.013708, 3.141563, -0.000000]),accel_mss,speed_ms,0,0.001)
      movel(pose_trans(ref_frame,p[0.139334, 0.016668, -0.000125, -0.013708, 3.141563, -0.000000]),accel_mss,speed_ms,0,0.001)
      movel(pose_trans(ref_frame,p[0.139181, 0.016680, -0.000125, -0.013708, 3.141563, -0.000000]),accel_mss,speed_ms,0,0.001)
      movel(pose_trans(ref_frame,p[0.139028, 0.016698, -0.000125, -0.013708, 3.141563, 0.000000]),accel_mss,speed_ms,0,0.001)
      movel(pose_trans(ref_frame,p[0.138904, 0.016717, -0.000125, -0.013708, 3.141563, -0.000000]),accel_mss,speed_ms,0,0.001)
      movel(pose_trans(ref_frame,p[0.138780, 0.016740, -0.000125, -0.013708, 3.141563, -0.000000]),accel_mss,speed_ms,0,0.001)
      movel(pose_trans(ref_frame,p[0.138728, 0.016758, -0.000125, -0.013708, 3.141563, -0.000000]),accel_mss,speed_ms,0,0.001)
      movel(pose_trans(ref_frame,p[0.138685, 0.016791, -0.000125, -0.013708, 3.141563, -0.000000]),accel_mss,speed_ms,0,0.001)
      movel(pose_trans(ref_frame,p[0.138621, 0.016881, -0.000125, -0.013708, 3.141563, 0.000000]),accel_mss,speed_ms,0,0.001)
      movel(pose_trans(ref_frame,p[0.138593, 0.016988, -0.000125, -0.013708, 3.141563, 0.000000]),accel_mss,speed_ms,0,0.001)
      movel(pose_trans(ref_frame,p[0.138575, 0.017264, -0.000125, -0.013708, 3.141563, -0.000000]),accel_mss,speed_ms,0,0.001)
      movel(pose_trans(ref_frame,p[0.138566, 0.017540, -0.000125, -0.013708, 3.141563, -0.000000]),accel_mss,speed_ms,0,0.001)
      movel(pose_trans(ref_frame,p[0.138565, 0.017817, -0.000125, -0.013708, 3.141563, 0.000000]),accel_mss,speed_ms,0,0.001)
      movel(pose_trans(ref_frame,p[0.138574, 0.018094, -0.000125, -0.013708, 3.141563, -0.000000]),accel_mss,speed_ms,0,0.001)
      movel(pose_trans(ref_frame,p[0.138598, 0.018198, -0.000125, -0.013708, 3.141563, -0.000000]),accel_mss,speed_ms,0,0.001)
      movel(pose_trans(ref_frame,p[0.138658, 0.018286, -0.000125, -0.013708, 3.141563, -0.000000]),accel_mss,speed_ms,0,0.001)
      movel(pose_trans(ref_frame,p[0.138691, 0.018309, -0.000125, -0.013708, 3.141563, -0.000000]),accel_mss,speed_ms,0,0.001)
      movel(pose_trans(ref_frame,p[0.138730, 0.018321, -0.000125, -0.013708, 3.141563, -0.000000]),accel_mss,speed_ms,0,0.001)
      movel(pose_trans(ref_frame,p[0.138855, 0.018335, -0.000125, -0.013708, 3.141563, -0.000000]),accel_mss,speed_ms,0,0.001)
      movel(pose_trans(ref_frame,p[0.138982, 0.018348, -0.000125, -0.013708, 3.141563, 0.000000]),accel_mss,speed_ms,0,0.001)
      movel(pose_trans(ref_frame,p[0.139135, 0.018359, -0.000125, -0.013708, 3.141563, 0.000000]),accel_mss,speed_ms,0,0.001)
      movel(pose_trans(ref_frame,p[0.139288, 0.018366, -0.000125, -0.013708, 3.141563, 0.000000]),accel_mss,speed_ms,0,0.001)
      movel(pose_trans(ref_frame,p[0.139461, 0.018371, -0.000125, -0.013708, 3.141563, -0.000000]),accel_mss,speed_ms,0,0.001)
      movel(pose_trans(ref_frame,p[0.139635, 0.018372, -0.000125, -0.013708, 3.141563, -0.000000]),accel_mss,speed_ms,0,0.001)
      movel(pose_trans(ref_frame,p[0.140523, 0.018370, -0.000125, -0.013708, 3.141563, -0.000000]),accel_mss,speed_ms,0,0.001)
      movel(pose_trans(ref_frame,p[0.140523, 0.019477, -0.000125, -0.013708, 3.141563, 0.000000]),accel_mss,speed_ms,0,0.001)
      movel(pose_trans(ref_frame,p[0.140523, 0.020584, -0.000125, -0.013708, 3.141563, -0.000000]),accel_mss,speed_ms,0,0.001)
      movel(pose_trans(ref_frame,p[0.139425, 0.020579, -0.000125, -0.013708, 3.141563, 0.000000]),accel_mss,speed_ms,0,0.001)
      movel(pose_trans(ref_frame,p[0.138326, 0.020574, -0.000125, -0.013708, 3.141563, -0.000000]),accel_mss,speed_ms,0,0.001)
      movel(pose_trans(ref_frame,p[0.138300, 0.019665, -0.000125, -0.013708, 3.141563, -0.000000]),accel_mss,speed_ms,0,0.001)
      movel(pose_trans(ref_frame,p[0.138295, 0.019489, -0.000125, -0.013708, 3.141563, -0.000000]),accel_mss,speed_ms,0,0.001)
      movel(pose_trans(ref_frame,p[0.138287, 0.019313, -0.000125, -0.013708, 3.141563, -0.000000]),accel_mss,speed_ms,0,0.001)
      movel(pose_trans(ref_frame,p[0.138279, 0.019161, -0.000125, -0.013708, 3.141563, -0.000000]),accel_mss,speed_ms,0,0.001)
      movel(pose_trans(ref_frame,p[0.138269, 0.019009, -0.000125, -0.013708, 3.141563, -0.000000]),accel_mss,speed_ms,0,0.001)
      movel(pose_trans(ref_frame,p[0.138258, 0.018880, -0.000125, -0.013708, 3.141563, -0.000000]),accel_mss,speed_ms,0,0.001)
      movel(pose_trans(ref_frame,p[0.138247, 0.018751, -0.000125, -0.013708, 3.141563, -0.000000]),accel_mss,speed_ms,0,0.001)
      movel(pose_trans(ref_frame,p[0.138241, 0.018728, -0.000125, -0.013708, 3.141563, 0.000000]),accel_mss,speed_ms,0,0.001)
      movel(pose_trans(ref_frame,p[0.138228, 0.018708, -0.000125, -0.013708, 3.141563, -0.000000]),accel_mss,speed_ms,0,0.001)
      movel(pose_trans(ref_frame,p[0.138148, 0.018654, -0.000125, -0.013708, 3.141563, -0.000000]),accel_mss,speed_ms,0,0.001)
      movel(pose_trans(ref_frame,p[0.138053, 0.018633, -0.000125, -0.013708, 3.141563, -0.000000]),accel_mss,speed_ms,0,0.001)
      movel(pose_trans(ref_frame,p[0.137769, 0.018628, -0.000125, -0.013708, 3.141563, 0.000000]),accel_mss,speed_ms,0,0.001)
      movel(pose_trans(ref_frame,p[0.137485, 0.018630, -0.000125, -0.013708, 3.141563, -0.000000]),accel_mss,speed_ms,0,0.001)
      movel(pose_trans(ref_frame,p[0.137202, 0.018639, -0.000125, -0.013708, 3.141563, -0.000000]),accel_mss,speed_ms,0,0.001)
      movel(pose_trans(ref_frame,p[0.136919, 0.018654, -0.000125, -0.013708, 3.141563, -0.000000]),accel_mss,speed_ms,0,0.001)
      movel(pose_trans(ref_frame,p[0.136822, 0.018679, -0.000125, -0.013708, 3.141563, 0.000000]),accel_mss,speed_ms,0,0.001)
      movel(pose_trans(ref_frame,p[0.136739, 0.018736, -0.000125, -0.013708, 3.141563, -0.000000]),accel_mss,speed_ms,0,0.001)
      movel(pose_trans(ref_frame,p[0.136654, 0.018863, -0.000125, -0.013708, 3.141563, 0.000000]),accel_mss,speed_ms,0,0.001)
      movel(pose_trans(ref_frame,p[0.136622, 0.019012, -0.000125, -0.013708, 3.141563, -0.000000]),accel_mss,speed_ms,0,0.001)
      movel(pose_trans(ref_frame,p[0.136610, 0.019729, -0.000125, -0.013708, 3.141563, 0.000000]),accel_mss,speed_ms,0,0.001)
      movel(pose_trans(ref_frame,p[0.136605, 0.020447, -0.000125, -0.013708, 3.141563, -0.000000]),accel_mss,speed_ms,0,0.001)
      movel(pose_trans(ref_frame,p[0.136606, 0.021165, -0.000125, -0.013708, 3.141563, -0.000000]),accel_mss,speed_ms,0,0.001)
      movel(pose_trans(ref_frame,p[0.136614, 0.021882, -0.000125, -0.013708, 3.141563, -0.000000]),accel_mss,speed_ms,0,0.001)
      movel(pose_trans(ref_frame,p[0.136645, 0.022031, -0.000125, -0.013708, 3.141563, 0.000000]),accel_mss,speed_ms,0,0.001)
      movel(pose_trans(ref_frame,p[0.136730, 0.022157, -0.000125, -0.013708, 3.141563, -0.000000]),accel_mss,speed_ms,0,0.001)
      movel(pose_trans(ref_frame,p[0.136779, 0.022192, -0.000125, -0.013708, 3.141563, -0.000000]),accel_mss,speed_ms,0,0.001)
      movel(pose_trans(ref_frame,p[0.136838, 0.022207, -0.000125, -0.013708, 3.141563, -0.000000]),accel_mss,speed_ms,0,0.001)
      movel(pose_trans(ref_frame,p[0.137098, 0.022229, -0.000125, -0.013708, 3.141563, -0.000000]),accel_mss,speed_ms,0,0.001)
      movel(pose_trans(ref_frame,p[0.137359, 0.022248, -0.000125, -0.013708, 3.141563, -0.000000]),accel_mss,speed_ms,0,0.001)
      movel(pose_trans(ref_frame,p[0.137670, 0.022266, -0.000125, -0.013708, 3.141563, -0.000000]),accel_mss,speed_ms,0,0.001)
      movel(pose_trans(ref_frame,p[0.137981, 0.022278, -0.000125, -0.013708, 3.141563, -0.000000]),accel_mss,speed_ms,0,0.001)
      movel(pose_trans(ref_frame,p[0.138339, 0.022286, -0.000125, -0.013708, 3.141563, -0.000000]),accel_mss,speed_ms,0,0.001)
      movel(pose_trans(ref_frame,p[0.138696, 0.022290, -0.000125, -0.013708, 3.141563, 0.000000]),accel_mss,speed_ms,0,0.001)
      movel(pose_trans(ref_frame,p[0.140537, 0.022297, -0.000125, -0.013708, 3.141563, -0.000000]),accel_mss,speed_ms,0,0.001)
      movel(pose_trans(ref_frame,p[0.140489, 0.056704, -0.000125, -0.013708, 3.141563, -0.000000]),accel_mss,speed_ms,0,0.001)
      movel(pose_trans(ref_frame,p[0.140480, 0.063951, -0.000125, -0.013708, 3.141563, -0.000000]),accel_mss,speed_ms,0,0.001)
      movel(pose_trans(ref_frame,p[0.140471, 0.071199, -0.000125, -0.013708, 3.141563, -0.000000]),accel_mss,speed_ms,0,0.001)
      movel(pose_trans(ref_frame,p[0.140463, 0.078750, -0.000125, -0.013708, 3.141563, 0.000000]),accel_mss,speed_ms,0,0.001)
      movel(pose_trans(ref_frame,p[0.140455, 0.086300, -0.000125, -0.013708, 3.141563, -0.000000]),accel_mss,speed_ms,0,0.001)
      movel(pose_trans(ref_frame,p[0.140449, 0.093103, -0.000125, -0.013708, 3.141563, -0.000000]),accel_mss,speed_ms,0,0.001)
      movel(pose_trans(ref_frame,p[0.140444, 0.099905, -0.000125, -0.013708, 3.141563, -0.000000]),accel_mss,speed_ms,0,0.001)
      movel(pose_trans(ref_frame,p[0.140441, 0.104524, -0.000125, -0.013708, 3.141563, 0.000000]),accel_mss,speed_ms,0,0.001)
      movel(pose_trans(ref_frame,p[0.140440, 0.109142, -0.000125, -0.013708, 3.141563, 0.000000]),accel_mss,speed_ms,0,0.001)
      movel(pose_trans(ref_frame,p[0.140440, 0.127174, -0.000125, -0.013708, 3.141563, 0.000000]),accel_mss,speed_ms,0,0.001)
      movel(pose_trans(ref_frame,p[0.138598, 0.127187, -0.000125, -0.013708, 3.141563, -0.000000]),accel_mss,speed_ms,0,0.001)
      movel(pose_trans(ref_frame,p[0.138241, 0.127192, -0.000125, -0.013708, 3.141563, -0.000000]),accel_mss,speed_ms,0,0.001)
      movel(pose_trans(ref_frame,p[0.137884, 0.127200, -0.000125, -0.013708, 3.141563, -0.000000]),accel_mss,speed_ms,0,0.001)
      movel(pose_trans(ref_frame,p[0.137575, 0.127212, -0.000125, -0.013708, 3.141563, 0.000000]),accel_mss,speed_ms,0,0.001)
      movel(pose_trans(ref_frame,p[0.137265, 0.127229, -0.000125, -0.013708, 3.141563, 0.000000]),accel_mss,speed_ms,0,0.001)
      movel(pose_trans(ref_frame,p[0.137004, 0.127246, -0.000125, -0.013708, 3.141563, 0.000000]),accel_mss,speed_ms,0,0.001)
      movel(pose_trans(ref_frame,p[0.136743, 0.127266, -0.000125, -0.013708, 3.141563, 0.000000]),accel_mss,speed_ms,0,0.001)
      movel(pose_trans(ref_frame,p[0.136691, 0.127279, -0.000125, -0.013708, 3.141563, -0.000000]),accel_mss,speed_ms,0,0.001)
      movel(pose_trans(ref_frame,p[0.136647, 0.127310, -0.000125, -0.013708, 3.141563, -0.000000]),accel_mss,speed_ms,0,0.001)
      movel(pose_trans(ref_frame,p[0.136567, 0.127429, -0.000125, -0.013708, 3.141563, -0.000000]),accel_mss,speed_ms,0,0.001)
      movel(pose_trans(ref_frame,p[0.136537, 0.127569, -0.000125, -0.013708, 3.141563, -0.000000]),accel_mss,speed_ms,0,0.001)
      movel(pose_trans(ref_frame,p[0.136528, 0.128292, -0.000125, -0.013708, 3.141563, -0.000000]),accel_mss,speed_ms,0,0.001)
      movel(pose_trans(ref_frame,p[0.136524, 0.129016, -0.000125, -0.013708, 3.141563, -0.000000]),accel_mss,speed_ms,0,0.001)
      movel(pose_trans(ref_frame,p[0.136527, 0.129739, -0.000125, -0.013708, 3.141563, 0.000000]),accel_mss,speed_ms,0,0.001)
      movel(pose_trans(ref_frame,p[0.136535, 0.130463, -0.000125, -0.013708, 3.141563, 0.000000]),accel_mss,speed_ms,0,0.001)
      movel(pose_trans(ref_frame,p[0.136564, 0.130603, -0.000125, -0.013708, 3.141563, 0.000000]),accel_mss,speed_ms,0,0.001)
      movel(pose_trans(ref_frame,p[0.136644, 0.130721, -0.000125, -0.013708, 3.141563, 0.000000]),accel_mss,speed_ms,0,0.001)
      movel(pose_trans(ref_frame,p[0.136735, 0.130785, -0.000125, -0.013708, 3.141563, 0.000000]),accel_mss,speed_ms,0,0.001)
      movel(pose_trans(ref_frame,p[0.136842, 0.130814, -0.000125, -0.013708, 3.141563, -0.000000]),accel_mss,speed_ms,0,0.001)
      movel(pose_trans(ref_frame,p[0.137118, 0.130836, -0.000125, -0.013708, 3.141563, 0.000000]),accel_mss,speed_ms,0,0.001)
      movel(pose_trans(ref_frame,p[0.137394, 0.130848, -0.000125, -0.013708, 3.141563, 0.000000]),accel_mss,speed_ms,0,0.001)
      movel(pose_trans(ref_frame,p[0.137672, 0.130852, -0.000125, -0.013708, 3.141563, -0.000000]),accel_mss,speed_ms,0,0.001)
      movel(pose_trans(ref_frame,p[0.137949, 0.130847, -0.000125, -0.013708, 3.141563, -0.000000]),accel_mss,speed_ms,0,0.001)
      movel(pose_trans(ref_frame,p[0.138052, 0.130824, -0.000125, -0.013708, 3.141563, 0.000000]),accel_mss,speed_ms,0,0.001)
      movel(pose_trans(ref_frame,p[0.138139, 0.130764, -0.000125, -0.013708, 3.141563, -0.000000]),accel_mss,speed_ms,0,0.001)
      movel(pose_trans(ref_frame,p[0.138160, 0.130734, -0.000125, -0.013708, 3.141563, 0.000000]),accel_mss,speed_ms,0,0.001)
      movel(pose_trans(ref_frame,p[0.138170, 0.130699, -0.000125, -0.013708, 3.141563, 0.000000]),accel_mss,speed_ms,0,0.001)
      movel(pose_trans(ref_frame,p[0.138184, 0.130572, -0.000125, -0.013708, 3.141563, 0.000000]),accel_mss,speed_ms,0,0.001)
      movel(pose_trans(ref_frame,p[0.138196, 0.130446, -0.000125, -0.013708, 3.141563, 0.000000]),accel_mss,speed_ms,0,0.001)
      movel(pose_trans(ref_frame,p[0.138208, 0.130292, -0.000125, -0.013708, 3.141563, 0.000000]),accel_mss,speed_ms,0,0.001)
      movel(pose_trans(ref_frame,p[0.138216, 0.130139, -0.000125, -0.013708, 3.141563, -0.000000]),accel_mss,speed_ms,0,0.001)
      movel(pose_trans(ref_frame,p[0.138221, 0.129964, -0.000125, -0.013708, 3.141563, 0.000000]),accel_mss,speed_ms,0,0.001)
      movel(pose_trans(ref_frame,p[0.138224, 0.129790, -0.000125, -0.013708, 3.141563, 0.000000]),accel_mss,speed_ms,0,0.001)
      movel(pose_trans(ref_frame,p[0.138229, 0.128894, -0.000125, -0.013708, 3.141563, -0.000000]),accel_mss,speed_ms,0,0.001)
      movel(pose_trans(ref_frame,p[0.139247, 0.128889, -0.000125, -0.013708, 3.141563, 0.000000]),accel_mss,speed_ms,0,0.001)
      movel(pose_trans(ref_frame,p[0.139445, 0.128890, -0.000125, -0.013708, 3.141563, 0.000000]),accel_mss,speed_ms,0,0.001)
      movel(pose_trans(ref_frame,p[0.139643, 0.128894, -0.000125, -0.013708, 3.141563, -0.000000]),accel_mss,speed_ms,0,0.001)
      movel(pose_trans(ref_frame,p[0.139818, 0.128901, -0.000125, -0.013708, 3.141563, 0.000000]),accel_mss,speed_ms,0,0.001)
      movel(pose_trans(ref_frame,p[0.139992, 0.128912, -0.000125, -0.013708, 3.141563, -0.000000]),accel_mss,speed_ms,0,0.001)
      movel(pose_trans(ref_frame,p[0.140137, 0.128924, -0.000125, -0.013708, 3.141563, 0.000000]),accel_mss,speed_ms,0,0.001)
      movel(pose_trans(ref_frame,p[0.140281, 0.128939, -0.000125, -0.013708, 3.141563, -0.000000]),accel_mss,speed_ms,0,0.001)
      movel(pose_trans(ref_frame,p[0.140321, 0.128950, -0.000125, -0.013708, 3.141563, 0.000000]),accel_mss,speed_ms,0,0.001)
      movel(pose_trans(ref_frame,p[0.140355, 0.128974, -0.000125, -0.013708, 3.141563, -0.000000]),accel_mss,speed_ms,0,0.001)
      movel(pose_trans(ref_frame,p[0.140380, 0.129009, -0.000125, -0.013708, 3.141563, 0.000000]),accel_mss,speed_ms,0,0.001)
      movel(pose_trans(ref_frame,p[0.140391, 0.129049, -0.000125, -0.013708, 3.141563, 0.000000]),accel_mss,speed_ms,0,0.001)
      movel(pose_trans(ref_frame,p[0.140406, 0.129193, -0.000125, -0.013708, 3.141563, 0.000000]),accel_mss,speed_ms,0,0.001)
      movel(pose_trans(ref_frame,p[0.140418, 0.129337, -0.000125, -0.013708, 3.141563, -0.000000]),accel_mss,speed_ms,0,0.001)
      movel(pose_trans(ref_frame,p[0.140429, 0.129512, -0.000125, -0.013708, 3.141563, 0.000000]),accel_mss,speed_ms,0,0.001)
      movel(pose_trans(ref_frame,p[0.140436, 0.129686, -0.000125, -0.013708, 3.141563, 0.000000]),accel_mss,speed_ms,0,0.001)
      movel(pose_trans(ref_frame,p[0.140440, 0.129885, -0.000125, -0.013708, 3.141563, 0.000000]),accel_mss,speed_ms,0,0.001)
      movel(pose_trans(ref_frame,p[0.140441, 0.130083, -0.000125, -0.013708, 3.141563, -0.000000]),accel_mss,speed_ms,0,0.001)
      movel(pose_trans(ref_frame,p[0.140435, 0.131101, -0.000125, -0.013708, 3.141563, 0.000000]),accel_mss,speed_ms,0,0.001)
      movel(pose_trans(ref_frame,p[0.139540, 0.131106, -0.000125, -0.013708, 3.141563, -0.000000]),accel_mss,speed_ms,0,0.001)
      movel(pose_trans(ref_frame,p[0.139365, 0.131109, -0.000125, -0.013708, 3.141563, 0.000000]),accel_mss,speed_ms,0,0.001)
      movel(pose_trans(ref_frame,p[0.139191, 0.131115, -0.000125, -0.013708, 3.141563, 0.000000]),accel_mss,speed_ms,0,0.001)
      movel(pose_trans(ref_frame,p[0.139036, 0.131123, -0.000125, -0.013708, 3.141563, 0.000000]),accel_mss,speed_ms,0,0.001)
      movel(pose_trans(ref_frame,p[0.138882, 0.131136, -0.000125, -0.013708, 3.141563, -0.000000]),accel_mss,speed_ms,0,0.001)
      movel(pose_trans(ref_frame,p[0.138755, 0.131149, -0.000125, -0.013708, 3.141563, -0.000000]),accel_mss,speed_ms,0,0.001)
      movel(pose_trans(ref_frame,p[0.138628, 0.131164, -0.000125, -0.013708, 3.141563, 0.000000]),accel_mss,speed_ms,0,0.001)
      movel(pose_trans(ref_frame,p[0.138590, 0.131175, -0.000125, -0.013708, 3.141563, 0.000000]),accel_mss,speed_ms,0,0.001)
      movel(pose_trans(ref_frame,p[0.138558, 0.131198, -0.000125, -0.013708, 3.141563, -0.000000]),accel_mss,speed_ms,0,0.001)
      movel(pose_trans(ref_frame,p[0.138500, 0.131284, -0.000125, -0.013708, 3.141563, -0.000000]),accel_mss,speed_ms,0,0.001)
      movel(pose_trans(ref_frame,p[0.138478, 0.131386, -0.000125, -0.013708, 3.141563, 0.000000]),accel_mss,speed_ms,0,0.001)
      movel(pose_trans(ref_frame,p[0.138476, 0.131664, -0.000125, -0.013708, 3.141563, 0.000000]),accel_mss,speed_ms,0,0.001)
      movel(pose_trans(ref_frame,p[0.138482, 0.131941, -0.000125, -0.013708, 3.141563, 0.000000]),accel_mss,speed_ms,0,0.001)
      movel(pose_trans(ref_frame,p[0.138497, 0.132218, -0.000125, -0.013708, 3.141563, -0.000000]),accel_mss,speed_ms,0,0.001)
      movel(pose_trans(ref_frame,p[0.138520, 0.132493, -0.000125, -0.013708, 3.141563, 0.000000]),accel_mss,speed_ms,0,0.001)
      movel(pose_trans(ref_frame,p[0.138550, 0.132601, -0.000125, -0.013708, 3.141563, -0.000000]),accel_mss,speed_ms,0,0.001)
      movel(pose_trans(ref_frame,p[0.138614, 0.132691, -0.000125, -0.013708, 3.141563, 0.000000]),accel_mss,speed_ms,0,0.001)
      movel(pose_trans(ref_frame,p[0.138656, 0.132723, -0.000125, -0.013708, 3.141563, -0.000000]),accel_mss,speed_ms,0,0.001)
      movel(pose_trans(ref_frame,p[0.138705, 0.132741, -0.000125, -0.013708, 3.141563, 0.000000]),accel_mss,speed_ms,0,0.001)
      movel(pose_trans(ref_frame,p[0.138816, 0.132762, -0.000125, -0.013708, 3.141563, 0.000000]),accel_mss,speed_ms,0,0.001)
      movel(pose_trans(ref_frame,p[0.138928, 0.132780, -0.000125, -0.013708, 3.141563, -0.000000]),accel_mss,speed_ms,0,0.001)
      movel(pose_trans(ref_frame,p[0.139065, 0.132795, -0.000125, -0.013708, 3.141563, -0.000000]),accel_mss,speed_ms,0,0.001)
      movel(pose_trans(ref_frame,p[0.139202, 0.132806, -0.000125, -0.013708, 3.141563, -0.000000]),accel_mss,speed_ms,0,0.001)
      movel(pose_trans(ref_frame,p[0.139352, 0.132811, -0.000125, -0.013708, 3.141563, 0.000000]),accel_mss,speed_ms,0,0.001)
      movel(pose_trans(ref_frame,p[0.139502, 0.132812, -0.000125, -0.013708, 3.141563, 0.000000]),accel_mss,speed_ms,0,0.001)
      movel(pose_trans(ref_frame,p[0.139651, 0.132812, -0.000125, -0.013708, 3.141563, 0.000000]),accel_mss,speed_ms,0,0.001)
      movel(pose_trans(ref_frame,p[0.139800, 0.132816, -0.000125, -0.013708, 3.141563, -0.000000]),accel_mss,speed_ms,0,0.001)
      movel(pose_trans(ref_frame,p[0.139934, 0.132823, -0.000125, -0.013708, 3.141563, 0.000000]),accel_mss,speed_ms,0,0.001)
      movel(pose_trans(ref_frame,p[0.140066, 0.132834, -0.000125, -0.013708, 3.141563, -0.000000]),accel_mss,speed_ms,0,0.001)
      movel(pose_trans(ref_frame,p[0.140175, 0.132846, -0.000125, -0.013708, 3.141563, 0.000000]),accel_mss,speed_ms,0,0.001)
      movel(pose_trans(ref_frame,p[0.140283, 0.132861, -0.000125, -0.013708, 3.141563, -0.000000]),accel_mss,speed_ms,0,0.001)
      movel(pose_trans(ref_frame,p[0.140322, 0.132873, -0.000125, -0.013708, 3.141563, 0.000000]),accel_mss,speed_ms,0,0.001)
      movel(pose_trans(ref_frame,p[0.140354, 0.132897, -0.000125, -0.013708, 3.141563, 0.000000]),accel_mss,speed_ms,0,0.001)
      movel(pose_trans(ref_frame,p[0.140379, 0.132931, -0.000125, -0.013708, 3.141563, -0.000000]),accel_mss,speed_ms,0,0.001)
      movel(pose_trans(ref_frame,p[0.140391, 0.132972, -0.000125, -0.013708, 3.141563, 0.000000]),accel_mss,speed_ms,0,0.001)
      movel(pose_trans(ref_frame,p[0.140405, 0.133116, -0.000125, -0.013708, 3.141563, -0.000000]),accel_mss,speed_ms,0,0.001)
      movel(pose_trans(ref_frame,p[0.140417, 0.133260, -0.000125, -0.013708, 3.141563, -0.000000]),accel_mss,speed_ms,0,0.001)
      movel(pose_trans(ref_frame,p[0.140429, 0.133435, -0.000125, -0.013708, 3.141563, -0.000000]),accel_mss,speed_ms,0,0.001)
      movel(pose_trans(ref_frame,p[0.140436, 0.133609, -0.000125, -0.013708, 3.141563, -0.000000]),accel_mss,speed_ms,0,0.001)
      movel(pose_trans(ref_frame,p[0.140440, 0.133808, -0.000125, -0.013708, 3.141563, 0.000000]),accel_mss,speed_ms,0,0.001)
      movel(pose_trans(ref_frame,p[0.140441, 0.134006, -0.000125, -0.013708, 3.141563, -0.000000]),accel_mss,speed_ms,0,0.001)
      movel(pose_trans(ref_frame,p[0.140435, 0.135024, -0.000125, -0.013708, 3.141563, 0.000000]),accel_mss,speed_ms,0,0.001)
      movel(pose_trans(ref_frame,p[0.139540, 0.135029, -0.000125, -0.013708, 3.141563, 0.000000]),accel_mss,speed_ms,0,0.001)
      movel(pose_trans(ref_frame,p[0.139365, 0.135032, -0.000125, -0.013708, 3.141563, 0.000000]),accel_mss,speed_ms,0,0.001)
      movel(pose_trans(ref_frame,p[0.139191, 0.135037, -0.000125, -0.013708, 3.141563, -0.000000]),accel_mss,speed_ms,0,0.001)
      movel(pose_trans(ref_frame,p[0.139037, 0.135045, -0.000125, -0.013708, 3.141563, -0.000000]),accel_mss,speed_ms,0,0.001)
      movel(pose_trans(ref_frame,p[0.138884, 0.135057, -0.000125, -0.013708, 3.141563, -0.000000]),accel_mss,speed_ms,0,0.001)
      movel(pose_trans(ref_frame,p[0.138757, 0.135069, -0.000125, -0.013708, 3.141563, 0.000000]),accel_mss,speed_ms,0,0.001)
      movel(pose_trans(ref_frame,p[0.138630, 0.135083, -0.000125, -0.013708, 3.141563, -0.000000]),accel_mss,speed_ms,0,0.001)
      movel(pose_trans(ref_frame,p[0.138595, 0.135093, -0.000125, -0.013708, 3.141563, 0.000000]),accel_mss,speed_ms,0,0.001)
      movel(pose_trans(ref_frame,p[0.138564, 0.135115, -0.000125, -0.013708, 3.141563, 0.000000]),accel_mss,speed_ms,0,0.001)
      movel(pose_trans(ref_frame,p[0.138543, 0.135145, -0.000125, -0.013708, 3.141563, 0.000000]),accel_mss,speed_ms,0,0.001)
      movel(pose_trans(ref_frame,p[0.138533, 0.135181, -0.000125, -0.013708, 3.141563, 0.000000]),accel_mss,speed_ms,0,0.001)
      movel(pose_trans(ref_frame,p[0.138519, 0.135307, -0.000125, -0.013708, 3.141563, 0.000000]),accel_mss,speed_ms,0,0.001)
      movel(pose_trans(ref_frame,p[0.138506, 0.135434, -0.000125, -0.013708, 3.141563, 0.000000]),accel_mss,speed_ms,0,0.001)
      movel(pose_trans(ref_frame,p[0.138495, 0.135588, -0.000125, -0.013708, 3.141563, 0.000000]),accel_mss,speed_ms,0,0.001)
      movel(pose_trans(ref_frame,p[0.138487, 0.135741, -0.000125, -0.013708, 3.141563, 0.000000]),accel_mss,speed_ms,0,0.001)
      movel(pose_trans(ref_frame,p[0.138481, 0.135916, -0.000125, -0.013708, 3.141563, 0.000000]),accel_mss,speed_ms,0,0.001)
      movel(pose_trans(ref_frame,p[0.138479, 0.136090, -0.000125, -0.013708, 3.141563, 0.000000]),accel_mss,speed_ms,0,0.001)
      movel(pose_trans(ref_frame,p[0.138473, 0.136986, -0.000125, -0.013708, 3.141563, -0.000000]),accel_mss,speed_ms,0,0.001)
      movel(pose_trans(ref_frame,p[0.137441, 0.136976, -0.000125, -0.013708, 3.141563, 0.000000]),accel_mss,speed_ms,0,0.001)
      movel(pose_trans(ref_frame,p[0.137240, 0.136973, -0.000125, -0.013708, 3.141563, 0.000000]),accel_mss,speed_ms,0,0.001)
      movel(pose_trans(ref_frame,p[0.137039, 0.136967, -0.000125, -0.013708, 3.141563, 0.000000]),accel_mss,speed_ms,0,0.001)
      movel(pose_trans(ref_frame,p[0.136864, 0.136959, -0.000125, -0.013708, 3.141563, 0.000000]),accel_mss,speed_ms,0,0.001)
      movel(pose_trans(ref_frame,p[0.136689, 0.136947, -0.000125, -0.013708, 3.141563, 0.000000]),accel_mss,speed_ms,0,0.001)
      movel(pose_trans(ref_frame,p[0.136542, 0.136935, -0.000125, -0.013708, 3.141563, 0.000000]),accel_mss,speed_ms,0,0.001)
      movel(pose_trans(ref_frame,p[0.136396, 0.136921, -0.000125, -0.013708, 3.141563, 0.000000]),accel_mss,speed_ms,0,0.001)
      movel(pose_trans(ref_frame,p[0.136361, 0.136911, -0.000125, -0.013708, 3.141563, 0.000000]),accel_mss,speed_ms,0,0.001)
      movel(pose_trans(ref_frame,p[0.136331, 0.136890, -0.000125, -0.013708, 3.141563, 0.000000]),accel_mss,speed_ms,0,0.001)
      movel(pose_trans(ref_frame,p[0.136311, 0.136862, -0.000125, -0.013708, 3.141563, -0.000000]),accel_mss,speed_ms,0,0.001)
      movel(pose_trans(ref_frame,p[0.136301, 0.136828, -0.000125, -0.013708, 3.141563, -0.000000]),accel_mss,speed_ms,0,0.001)
      movel(pose_trans(ref_frame,p[0.136289, 0.136720, -0.000125, -0.013708, 3.141563, -0.000000]),accel_mss,speed_ms,0,0.001)
      movel(pose_trans(ref_frame,p[0.136279, 0.136612, -0.000125, -0.013708, 3.141563, -0.000000]),accel_mss,speed_ms,0,0.001)
      movel(pose_trans(ref_frame,p[0.136270, 0.136481, -0.000125, -0.013708, 3.141563, -0.000000]),accel_mss,speed_ms,0,0.001)
      movel(pose_trans(ref_frame,p[0.136265, 0.136350, -0.000125, -0.013708, 3.141563, -0.000000]),accel_mss,speed_ms,0,0.001)
      movel(pose_trans(ref_frame,p[0.136262, 0.136201, -0.000125, -0.013708, 3.141563, -0.000000]),accel_mss,speed_ms,0,0.001)
      movel(pose_trans(ref_frame,p[0.136262, 0.136053, -0.000125, -0.013708, 3.141563, -0.000000]),accel_mss,speed_ms,0,0.001)
      movel(pose_trans(ref_frame,p[0.136261, 0.135902, -0.000125, -0.013708, 3.141563, -0.000000]),accel_mss,speed_ms,0,0.001)
      movel(pose_trans(ref_frame,p[0.136255, 0.135752, -0.000125, -0.013708, 3.141563, 0.000000]),accel_mss,speed_ms,0,0.001)
      movel(pose_trans(ref_frame,p[0.136244, 0.135614, -0.000125, -0.013708, 3.141563, -0.000000]),accel_mss,speed_ms,0,0.001)
      movel(pose_trans(ref_frame,p[0.136227, 0.135476, -0.000125, -0.013708, 3.141563, 0.000000]),accel_mss,speed_ms,0,0.001)
      movel(pose_trans(ref_frame,p[0.136209, 0.135364, -0.000125, -0.013708, 3.141563, 0.000000]),accel_mss,speed_ms,0,0.001)
      movel(pose_trans(ref_frame,p[0.136186, 0.135252, -0.000125, -0.013708, 3.141563, 0.000000]),accel_mss,speed_ms,0,0.001)
      movel(pose_trans(ref_frame,p[0.136167, 0.135201, -0.000125, -0.013708, 3.141563, -0.000000]),accel_mss,speed_ms,0,0.001)
      movel(pose_trans(ref_frame,p[0.136134, 0.135157, -0.000125, -0.013708, 3.141563, -0.000000]),accel_mss,speed_ms,0,0.001)
      movel(pose_trans(ref_frame,p[0.136043, 0.135094, -0.000125, -0.013708, 3.141563, 0.000000]),accel_mss,speed_ms,0,0.001)
      movel(pose_trans(ref_frame,p[0.135937, 0.135065, -0.000125, -0.013708, 3.141563, -0.000000]),accel_mss,speed_ms,0,0.001)
      movel(pose_trans(ref_frame,p[0.135661, 0.135044, -0.000125, -0.013708, 3.141563, -0.000000]),accel_mss,speed_ms,0,0.001)
      movel(pose_trans(ref_frame,p[0.135384, 0.135032, -0.000125, -0.013708, 3.141563, -0.000000]),accel_mss,speed_ms,0,0.001)
      movel(pose_trans(ref_frame,p[0.135107, 0.135029, -0.000125, -0.013708, 3.141563, 0.000000]),accel_mss,speed_ms,0,0.001)
      movel(pose_trans(ref_frame,p[0.134830, 0.135034, -0.000125, -0.013708, 3.141563, 0.000000]),accel_mss,speed_ms,0,0.001)
      movel(pose_trans(ref_frame,p[0.134727, 0.135057, -0.000125, -0.013708, 3.141563, -0.000000]),accel_mss,speed_ms,0,0.001)
      movel(pose_trans(ref_frame,p[0.134641, 0.135116, -0.000125, -0.013708, 3.141563, 0.000000]),accel_mss,speed_ms,0,0.001)
      movel(pose_trans(ref_frame,p[0.134619, 0.135146, -0.000125, -0.013708, 3.141563, -0.000000]),accel_mss,speed_ms,0,0.001)
      movel(pose_trans(ref_frame,p[0.134609, 0.135181, -0.000125, -0.013708, 3.141563, -0.000000]),accel_mss,speed_ms,0,0.001)
      movel(pose_trans(ref_frame,p[0.134595, 0.135309, -0.000125, -0.013708, 3.141563, 0.000000]),accel_mss,speed_ms,0,0.001)
      movel(pose_trans(ref_frame,p[0.134583, 0.135437, -0.000125, -0.013708, 3.141563, 0.000000]),accel_mss,speed_ms,0,0.001)
      movel(pose_trans(ref_frame,p[0.134571, 0.135591, -0.000125, -0.013708, 3.141563, 0.000000]),accel_mss,speed_ms,0,0.001)
      movel(pose_trans(ref_frame,p[0.134563, 0.135746, -0.000125, -0.013708, 3.141563, -0.000000]),accel_mss,speed_ms,0,0.001)
      movel(pose_trans(ref_frame,p[0.134557, 0.135921, -0.000125, -0.013708, 3.141563, 0.000000]),accel_mss,speed_ms,0,0.001)
      movel(pose_trans(ref_frame,p[0.134555, 0.136097, -0.000125, -0.013708, 3.141563, -0.000000]),accel_mss,speed_ms,0,0.001)
      movel(pose_trans(ref_frame,p[0.134548, 0.136999, -0.000125, -0.013708, 3.141563, 0.000000]),accel_mss,speed_ms,0,0.001)
      movel(pose_trans(ref_frame,p[0.133508, 0.136975, -0.000125, -0.013708, 3.141563, 0.000000]),accel_mss,speed_ms,0,0.001)
      movel(pose_trans(ref_frame,p[0.133308, 0.136970, -0.000125, -0.013708, 3.141563, -0.000000]),accel_mss,speed_ms,0,0.001)
      movel(pose_trans(ref_frame,p[0.133107, 0.136963, -0.000125, -0.013708, 3.141563, 0.000000]),accel_mss,speed_ms,0,0.001)
      movel(pose_trans(ref_frame,p[0.132935, 0.136956, -0.000125, -0.013708, 3.141563, 0.000000]),accel_mss,speed_ms,0,0.001)
      movel(pose_trans(ref_frame,p[0.132763, 0.136947, -0.000125, -0.013708, 3.141563, -0.000000]),accel_mss,speed_ms,0,0.001)
      movel(pose_trans(ref_frame,p[0.132615, 0.136938, -0.000125, -0.013708, 3.141563, -0.000000]),accel_mss,speed_ms,0,0.001)
      movel(pose_trans(ref_frame,p[0.132466, 0.136929, -0.000125, -0.013708, 3.141563, 0.000000]),accel_mss,speed_ms,0,0.001)
      movel(pose_trans(ref_frame,p[0.132448, 0.136924, -0.000125, -0.013708, 3.141563, -0.000000]),accel_mss,speed_ms,0,0.001)
      movel(pose_trans(ref_frame,p[0.132432, 0.136914, -0.000125, -0.013708, 3.141563, -0.000000]),accel_mss,speed_ms,0,0.001)
      movel(pose_trans(ref_frame,p[0.132421, 0.136898, -0.000125, -0.013708, 3.141563, 0.000000]),accel_mss,speed_ms,0,0.001)
      movel(pose_trans(ref_frame,p[0.132417, 0.136880, -0.000125, -0.013708, 3.141563, -0.000000]),accel_mss,speed_ms,0,0.001)
      movel(pose_trans(ref_frame,p[0.132411, 0.136730, -0.000125, -0.013708, 3.141563, -0.000000]),accel_mss,speed_ms,0,0.001)
      movel(pose_trans(ref_frame,p[0.132406, 0.136581, -0.000125, -0.013708, 3.141563, 0.000000]),accel_mss,speed_ms,0,0.001)
      movel(pose_trans(ref_frame,p[0.132401, 0.136409, -0.000125, -0.013708, 3.141563, -0.000000]),accel_mss,speed_ms,0,0.001)
      movel(pose_trans(ref_frame,p[0.132398, 0.136236, -0.000125, -0.013708, 3.141563, 0.000000]),accel_mss,speed_ms,0,0.001)
      movel(pose_trans(ref_frame,p[0.132396, 0.136035, -0.000125, -0.013708, 3.141563, -0.000000]),accel_mss,speed_ms,0,0.001)
      movel(pose_trans(ref_frame,p[0.132395, 0.135834, -0.000125, -0.013708, 3.141563, -0.000000]),accel_mss,speed_ms,0,0.001)
      movel(pose_trans(ref_frame,p[0.132395, 0.134791, -0.000125, -0.013708, 3.141563, 0.000000]),accel_mss,speed_ms,0,0.001)
      movel(pose_trans(ref_frame,p[0.133279, 0.134766, -0.000125, -0.013708, 3.141563, 0.000000]),accel_mss,speed_ms,0,0.001)
      movel(pose_trans(ref_frame,p[0.133451, 0.134760, -0.000125, -0.013708, 3.141563, 0.000000]),accel_mss,speed_ms,0,0.001)
      movel(pose_trans(ref_frame,p[0.133623, 0.134751, -0.000125, -0.013708, 3.141563, 0.000000]),accel_mss,speed_ms,0,0.001)
      movel(pose_trans(ref_frame,p[0.133774, 0.134741, -0.000125, -0.013708, 3.141563, 0.000000]),accel_mss,speed_ms,0,0.001)
      movel(pose_trans(ref_frame,p[0.133924, 0.134727, -0.000125, -0.013708, 3.141563, 0.000000]),accel_mss,speed_ms,0,0.001)
      movel(pose_trans(ref_frame,p[0.134049, 0.134713, -0.000125, -0.013708, 3.141563, 0.000000]),accel_mss,speed_ms,0,0.001)
      movel(pose_trans(ref_frame,p[0.134174, 0.134698, -0.000125, -0.013708, 3.141563, 0.000000]),accel_mss,speed_ms,0,0.001)
      movel(pose_trans(ref_frame,p[0.134207, 0.134688, -0.000125, -0.013708, 3.141563, -0.000000]),accel_mss,speed_ms,0,0.001)
      movel(pose_trans(ref_frame,p[0.134235, 0.134668, -0.000125, -0.013708, 3.141563, 0.000000]),accel_mss,speed_ms,0,0.001)
      movel(pose_trans(ref_frame,p[0.134289, 0.134588, -0.000125, -0.013708, 3.141563, -0.000000]),accel_mss,speed_ms,0,0.001)
      movel(pose_trans(ref_frame,p[0.134309, 0.134492, -0.000125, -0.013708, 3.141563, -0.000000]),accel_mss,speed_ms,0,0.001)
      movel(pose_trans(ref_frame,p[0.134307, 0.134213, -0.000125, -0.013708, 3.141563, 0.000000]),accel_mss,speed_ms,0,0.001)
      movel(pose_trans(ref_frame,p[0.134298, 0.133934, -0.000125, -0.013708, 3.141563, 0.000000]),accel_mss,speed_ms,0,0.001)
      movel(pose_trans(ref_frame,p[0.134281, 0.133656, -0.000125, -0.013708, 3.141563, 0.000000]),accel_mss,speed_ms,0,0.001)
      movel(pose_trans(ref_frame,p[0.134257, 0.133379, -0.000125, -0.013708, 3.141563, -0.000000]),accel_mss,speed_ms,0,0.001)
      movel(pose_trans(ref_frame,p[0.134228, 0.133277, -0.000125, -0.013708, 3.141563, -0.000000]),accel_mss,speed_ms,0,0.001)
      movel(pose_trans(ref_frame,p[0.134167, 0.133191, -0.000125, -0.013708, 3.141563, -0.000000]),accel_mss,speed_ms,0,0.001)
      movel(pose_trans(ref_frame,p[0.134055, 0.133115, -0.000125, -0.013708, 3.141563, 0.000000]),accel_mss,speed_ms,0,0.001)
      movel(pose_trans(ref_frame,p[0.133921, 0.133086, -0.000125, -0.013708, 3.141563, -0.000000]),accel_mss,speed_ms,0,0.001)
      movel(pose_trans(ref_frame,p[0.133197, 0.133076, -0.000125, -0.013708, 3.141563, -0.000000]),accel_mss,speed_ms,0,0.001)
      movel(pose_trans(ref_frame,p[0.132473, 0.133070, -0.000125, -0.013708, 3.141563, 0.000000]),accel_mss,speed_ms,0,0.001)
      movel(pose_trans(ref_frame,p[0.131748, 0.133070, -0.000125, -0.013708, 3.141563, 0.000000]),accel_mss,speed_ms,0,0.001)
      movel(pose_trans(ref_frame,p[0.131024, 0.133075, -0.000125, -0.013708, 3.141563, 0.000000]),accel_mss,speed_ms,0,0.001)
      movel(pose_trans(ref_frame,p[0.130892, 0.133102, -0.000125, -0.013708, 3.141563, -0.000000]),accel_mss,speed_ms,0,0.001)
      movel(pose_trans(ref_frame,p[0.130779, 0.133178, -0.000125, -0.013708, 3.141563, 0.000000]),accel_mss,speed_ms,0,0.001)
      movel(pose_trans(ref_frame,p[0.130750, 0.133221, -0.000125, -0.013708, 3.141563, 0.000000]),accel_mss,speed_ms,0,0.001)
      movel(pose_trans(ref_frame,p[0.130736, 0.133271, -0.000125, -0.013708, 3.141563, 0.000000]),accel_mss,speed_ms,0,0.001)
      movel(pose_trans(ref_frame,p[0.130718, 0.133527, -0.000125, -0.013708, 3.141563, 0.000000]),accel_mss,speed_ms,0,0.001)
      movel(pose_trans(ref_frame,p[0.130701, 0.133784, -0.000125, -0.013708, 3.141563, 0.000000]),accel_mss,speed_ms,0,0.001)
      movel(pose_trans(ref_frame,p[0.130685, 0.134087, -0.000125, -0.013708, 3.141563, -0.000000]),accel_mss,speed_ms,0,0.001)
      movel(pose_trans(ref_frame,p[0.130674, 0.134391, -0.000125, -0.013708, 3.141563, -0.000000]),accel_mss,speed_ms,0,0.001)
      movel(pose_trans(ref_frame,p[0.130666, 0.134741, -0.000125, -0.013708, 3.141563, 0.000000]),accel_mss,speed_ms,0,0.001)
      movel(pose_trans(ref_frame,p[0.130662, 0.135091, -0.000125, -0.013708, 3.141563, 0.000000]),accel_mss,speed_ms,0,0.001)
      movel(pose_trans(ref_frame,p[0.130658, 0.135438, -0.000125, -0.013708, 3.141563, -0.000000]),accel_mss,speed_ms,0,0.001)
      movel(pose_trans(ref_frame,p[0.130652, 0.135786, -0.000125, -0.013708, 3.141563, 0.000000]),accel_mss,speed_ms,0,0.001)
      movel(pose_trans(ref_frame,p[0.130643, 0.136081, -0.000125, -0.013708, 3.141563, -0.000000]),accel_mss,speed_ms,0,0.001)
      movel(pose_trans(ref_frame,p[0.130630, 0.136377, -0.000125, -0.013708, 3.141563, -0.000000]),accel_mss,speed_ms,0,0.001)
      movel(pose_trans(ref_frame,p[0.130616, 0.136631, -0.000125, -0.013708, 3.141563, -0.000000]),accel_mss,speed_ms,0,0.001)
      movel(pose_trans(ref_frame,p[0.130602, 0.136885, -0.000125, -0.013708, 3.141563, 0.000000]),accel_mss,speed_ms,0,0.001)
      movel(pose_trans(ref_frame,p[0.130591, 0.136914, -0.000125, -0.013708, 3.141563, 0.000000]),accel_mss,speed_ms,0,0.001)
      movel(pose_trans(ref_frame,p[0.130568, 0.136933, -0.000125, -0.013708, 3.141563, 0.000000]),accel_mss,speed_ms,0,0.001)
      movel(pose_trans(ref_frame,p[0.130533, 0.136944, -0.000125, -0.013708, 3.141563, 0.000000]),accel_mss,speed_ms,0,0.001)
      movel(pose_trans(ref_frame,p[0.130496, 0.136948, -0.000125, -0.013708, 3.141563, -0.000000]),accel_mss,speed_ms,0,0.001)
      movel(pose_trans(ref_frame,p[0.115124, 0.136974, -0.000125, -0.013708, 3.141563, -0.000000]),accel_mss,speed_ms,0,0.001)
      movel(pose_trans(ref_frame,p[0.106662, 0.136988, -0.000125, -0.013708, 3.141563, 0.000000]),accel_mss,speed_ms,0,0.001)
      movel(pose_trans(ref_frame,p[0.098199, 0.136999, -0.000125, -0.013708, 3.141563, 0.000000]),accel_mss,speed_ms,0,0.001)
      movel(pose_trans(ref_frame,p[0.088155, 0.137011, -0.000125, -0.013708, 3.141563, 0.000000]),accel_mss,speed_ms,0,0.001)
      movel(pose_trans(ref_frame,p[0.078111, 0.137022, -0.000125, -0.013708, 3.141563, -0.000000]),accel_mss,speed_ms,0,0.001)
      movel(pose_trans(ref_frame,p[0.025738, 0.137075, -0.000125, -0.013708, 3.141563, 0.000000]),accel_mss,speed_ms,0,0.001)
      movel(pose_trans(ref_frame,p[0.025735, 0.135241, -0.000125, -0.013708, 3.141563, -0.000000]),accel_mss,speed_ms,0,0.001)
      movel(pose_trans(ref_frame,p[0.025732, 0.134884, -0.000125, -0.013708, 3.141563, -0.000000]),accel_mss,speed_ms,0,0.001)
      movel(pose_trans(ref_frame,p[0.025724, 0.134528, -0.000125, -0.013708, 3.141563, 0.000000]),accel_mss,speed_ms,0,0.001)
      movel(pose_trans(ref_frame,p[0.025713, 0.134218, -0.000125, -0.013708, 3.141563, 0.000000]),accel_mss,speed_ms,0,0.001)
      movel(pose_trans(ref_frame,p[0.025695, 0.133908, -0.000125, -0.013708, 3.141563, -0.000000]),accel_mss,speed_ms,0,0.001)
      movel(pose_trans(ref_frame,p[0.025676, 0.133648, -0.000125, -0.013708, 3.141563, 0.000000]),accel_mss,speed_ms,0,0.001)
      movel(pose_trans(ref_frame,p[0.025655, 0.133388, -0.000125, -0.013708, 3.141563, 0.000000]),accel_mss,speed_ms,0,0.001)
      movel(pose_trans(ref_frame,p[0.025639, 0.133329, -0.000125, -0.013708, 3.141563, 0.000000]),accel_mss,speed_ms,0,0.001)
      movel(pose_trans(ref_frame,p[0.025604, 0.133278, -0.000125, -0.013708, 3.141563, -0.000000]),accel_mss,speed_ms,0,0.001)
      movel(pose_trans(ref_frame,p[0.025480, 0.133195, -0.000125, -0.013708, 3.141563, -0.000000]),accel_mss,speed_ms,0,0.001)
      movel(pose_trans(ref_frame,p[0.025335, 0.133165, -0.000125, -0.013708, 3.141563, -0.000000]),accel_mss,speed_ms,0,0.001)
      movel(pose_trans(ref_frame,p[0.024616, 0.133157, -0.000125, -0.013708, 3.141563, -0.000000]),accel_mss,speed_ms,0,0.001)
      movel(pose_trans(ref_frame,p[0.023897, 0.133156, -0.000125, -0.013708, 3.141563, -0.000000]),accel_mss,speed_ms,0,0.001)
      movel(pose_trans(ref_frame,p[0.023178, 0.133161, -0.000125, -0.013708, 3.141563, 0.000000]),accel_mss,speed_ms,0,0.001)
      movel(pose_trans(ref_frame,p[0.022459, 0.133172, -0.000125, -0.013708, 3.141563, 0.000000]),accel_mss,speed_ms,0,0.001)
      movel(pose_trans(ref_frame,p[0.022313, 0.133204, -0.000125, -0.013708, 3.141563, -0.000000]),accel_mss,speed_ms,0,0.001)
      movel(pose_trans(ref_frame,p[0.022189, 0.133287, -0.000125, -0.013708, 3.141563, -0.000000]),accel_mss,speed_ms,0,0.001)
      movel(pose_trans(ref_frame,p[0.022117, 0.133391, -0.000125, -0.013708, 3.141563, 0.000000]),accel_mss,speed_ms,0,0.001)
      movel(pose_trans(ref_frame,p[0.022084, 0.133512, -0.000125, -0.013708, 3.141563, 0.000000]),accel_mss,speed_ms,0,0.001)
      movel(pose_trans(ref_frame,p[0.022070, 0.133748, -0.000125, -0.013708, 3.141563, 0.000000]),accel_mss,speed_ms,0,0.001)
      movel(pose_trans(ref_frame,p[0.022071, 0.133983, -0.000125, -0.013708, 3.141563, -0.000000]),accel_mss,speed_ms,0,0.001)
      movel(pose_trans(ref_frame,p[0.022087, 0.134220, -0.000125, -0.013708, 3.141563, 0.000000]),accel_mss,speed_ms,0,0.001)
      movel(pose_trans(ref_frame,p[0.022119, 0.134454, -0.000125, -0.013708, 3.141563, 0.000000]),accel_mss,speed_ms,0,0.001)
      movel(pose_trans(ref_frame,p[0.022160, 0.134581, -0.000125, -0.013708, 3.141563, -0.000000]),accel_mss,speed_ms,0,0.001)
      movel(pose_trans(ref_frame,p[0.022239, 0.134690, -0.000125, -0.013708, 3.141563, 0.000000]),accel_mss,speed_ms,0,0.001)
      movel(pose_trans(ref_frame,p[0.022291, 0.134729, -0.000125, -0.013708, 3.141563, 0.000000]),accel_mss,speed_ms,0,0.001)
      movel(pose_trans(ref_frame,p[0.022350, 0.134754, -0.000125, -0.013708, 3.141563, 0.000000]),accel_mss,speed_ms,0,0.001)
      movel(pose_trans(ref_frame,p[0.022471, 0.134783, -0.000125, -0.013708, 3.141563, -0.000000]),accel_mss,speed_ms,0,0.001)
      movel(pose_trans(ref_frame,p[0.022593, 0.134807, -0.000125, -0.013708, 3.141563, 0.000000]),accel_mss,speed_ms,0,0.001)
      movel(pose_trans(ref_frame,p[0.022741, 0.134829, -0.000125, -0.013708, 3.141563, 0.000000]),accel_mss,speed_ms,0,0.001)
      movel(pose_trans(ref_frame,p[0.022891, 0.134845, -0.000125, -0.013708, 3.141563, 0.000000]),accel_mss,speed_ms,0,0.001)
      movel(pose_trans(ref_frame,p[0.023052, 0.134855, -0.000125, -0.013708, 3.141563, 0.000000]),accel_mss,speed_ms,0,0.001)
      movel(pose_trans(ref_frame,p[0.023213, 0.134859, -0.000125, -0.013708, 3.141563, 0.000000]),accel_mss,speed_ms,0,0.001)
      movel(pose_trans(ref_frame,p[0.024024, 0.134865, -0.000125, -0.013708, 3.141563, 0.000000]),accel_mss,speed_ms,0,0.001)
      movel(pose_trans(ref_frame,p[0.024029, 0.135970, -0.000125, -0.013708, 3.141563, 0.000000]),accel_mss,speed_ms,0,0.001)
      movel(pose_trans(ref_frame,p[0.024034, 0.137075, -0.000125, -0.013708, 3.141563, -0.000000]),accel_mss,speed_ms,0,0.001)
      movel(pose_trans(ref_frame,p[0.022932, 0.137075, -0.000125, -0.013708, 3.141563, 0.000000]),accel_mss,speed_ms,0,0.001)
      movel(pose_trans(ref_frame,p[0.021829, 0.137075, -0.000125, -0.013708, 3.141563, 0.000000]),accel_mss,speed_ms,0,0.001)
      movel(pose_trans(ref_frame,p[0.021877, 0.136331, -0.000125, -0.013708, 3.141563, 0.000000]),accel_mss,speed_ms,0,0.001)
      movel(pose_trans(ref_frame,p[0.021890, 0.135997, -0.000125, -0.013708, 3.141563, -0.000000]),accel_mss,speed_ms,0,0.001)
      movel(pose_trans(ref_frame,p[0.021886, 0.135664, -0.000125, -0.013708, 3.141563, -0.000000]),accel_mss,speed_ms,0,0.001)
      movel(pose_trans(ref_frame,p[0.021855, 0.135492, -0.000125, -0.013708, 3.141563, 0.000000]),accel_mss,speed_ms,0,0.001)
      movel(pose_trans(ref_frame,p[0.021777, 0.135336, -0.000125, -0.013708, 3.141563, -0.000000]),accel_mss,speed_ms,0,0.001)
      movel(pose_trans(ref_frame,p[0.021666, 0.135228, -0.000125, -0.013708, 3.141563, -0.000000]),accel_mss,speed_ms,0,0.001)
      movel(pose_trans(ref_frame,p[0.021524, 0.135169, -0.000125, -0.013708, 3.141563, -0.000000]),accel_mss,speed_ms,0,0.001)
      movel(pose_trans(ref_frame,p[0.021277, 0.135130, -0.000125, -0.013708, 3.141563, -0.000000]),accel_mss,speed_ms,0,0.001)
      movel(pose_trans(ref_frame,p[0.021026, 0.135115, -0.000125, -0.013708, 3.141563, -0.000000]),accel_mss,speed_ms,0,0.001)
      movel(pose_trans(ref_frame,p[0.020896, 0.135115, -0.000125, -0.013708, 3.141563, 0.000000]),accel_mss,speed_ms,0,0.001)
      movel(pose_trans(ref_frame,p[0.020766, 0.135121, -0.000125, -0.013708, 3.141563, 0.000000]),accel_mss,speed_ms,0,0.001)
      movel(pose_trans(ref_frame,p[0.020646, 0.135130, -0.000125, -0.013708, 3.141563, 0.000000]),accel_mss,speed_ms,0,0.001)
      movel(pose_trans(ref_frame,p[0.020527, 0.135145, -0.000125, -0.013708, 3.141563, 0.000000]),accel_mss,speed_ms,0,0.001)
      movel(pose_trans(ref_frame,p[0.020430, 0.135161, -0.000125, -0.013708, 3.141563, 0.000000]),accel_mss,speed_ms,0,0.001)
      movel(pose_trans(ref_frame,p[0.020333, 0.135181, -0.000125, -0.013708, 3.141563, 0.000000]),accel_mss,speed_ms,0,0.001)
      movel(pose_trans(ref_frame,p[0.020288, 0.135199, -0.000125, -0.013708, 3.141563, 0.000000]),accel_mss,speed_ms,0,0.001)
      movel(pose_trans(ref_frame,p[0.020249, 0.135228, -0.000125, -0.013708, 3.141563, 0.000000]),accel_mss,speed_ms,0,0.001)
      movel(pose_trans(ref_frame,p[0.020218, 0.135270, -0.000125, -0.013708, 3.141563, 0.000000]),accel_mss,speed_ms,0,0.001)
      movel(pose_trans(ref_frame,p[0.020202, 0.135319, -0.000125, -0.013708, 3.141563, 0.000000]),accel_mss,speed_ms,0,0.001)
      movel(pose_trans(ref_frame,p[0.020183, 0.135442, -0.000125, -0.013708, 3.141563, 0.000000]),accel_mss,speed_ms,0,0.001)
      movel(pose_trans(ref_frame,p[0.020167, 0.135567, -0.000125, -0.013708, 3.141563, 0.000000]),accel_mss,speed_ms,0,0.001)
      movel(pose_trans(ref_frame,p[0.020153, 0.135719, -0.000125, -0.013708, 3.141563, -0.000000]),accel_mss,speed_ms,0,0.001)
      movel(pose_trans(ref_frame,p[0.020145, 0.135872, -0.000125, -0.013708, 3.141563, -0.000000]),accel_mss,speed_ms,0,0.001)
      movel(pose_trans(ref_frame,p[0.020141, 0.136041, -0.000125, -0.013708, 3.141563, -0.000000]),accel_mss,speed_ms,0,0.001)
      movel(pose_trans(ref_frame,p[0.020141, 0.136210, -0.000125, -0.013708, 3.141563, -0.000000]),accel_mss,speed_ms,0,0.001)
      movel(pose_trans(ref_frame,p[0.020155, 0.137072, -0.000125, -0.013708, 3.141563, 0.000000]),accel_mss,speed_ms,0,0.001)
      movel(pose_trans(ref_frame,p[0.019067, 0.137076, -0.000125, -0.013708, 3.141563, 0.000000]),accel_mss,speed_ms,0,0.001)
      movel(pose_trans(ref_frame,p[0.017979, 0.137081, -0.000125, -0.013708, 3.141563, 0.000000]),accel_mss,speed_ms,0,0.001)
      movel(pose_trans(ref_frame,p[0.017974, 0.136223, -0.000125, -0.013708, 3.141563, -0.000000]),accel_mss,speed_ms,0,0.001)
      movel(pose_trans(ref_frame,p[0.017971, 0.136054, -0.000125, -0.013708, 3.141563, -0.000000]),accel_mss,speed_ms,0,0.001)
      movel(pose_trans(ref_frame,p[0.017963, 0.135886, -0.000125, -0.013708, 3.141563, 0.000000]),accel_mss,speed_ms,0,0.001)
      movel(pose_trans(ref_frame,p[0.017951, 0.135733, -0.000125, -0.013708, 3.141563, 0.000000]),accel_mss,speed_ms,0,0.001)
      movel(pose_trans(ref_frame,p[0.017934, 0.135581, -0.000125, -0.013708, 3.141563, -0.000000]),accel_mss,speed_ms,0,0.001)
      movel(pose_trans(ref_frame,p[0.017916, 0.135457, -0.000125, -0.013708, 3.141563, 0.000000]),accel_mss,speed_ms,0,0.001)
      movel(pose_trans(ref_frame,p[0.017894, 0.135334, -0.000125, -0.013708, 3.141563, 0.000000]),accel_mss,speed_ms,0,0.001)
      movel(pose_trans(ref_frame,p[0.017877, 0.135285, -0.000125, -0.013708, 3.141563, 0.000000]),accel_mss,speed_ms,0,0.001)
      movel(pose_trans(ref_frame,p[0.017846, 0.135243, -0.000125, -0.013708, 3.141563, -0.000000]),accel_mss,speed_ms,0,0.001)
      movel(pose_trans(ref_frame,p[0.017804, 0.135212, -0.000125, -0.013708, 3.141563, -0.000000]),accel_mss,speed_ms,0,0.001)
      movel(pose_trans(ref_frame,p[0.017755, 0.135194, -0.000125, -0.013708, 3.141563, 0.000000]),accel_mss,speed_ms,0,0.001)
      movel(pose_trans(ref_frame,p[0.017631, 0.135173, -0.000125, -0.013708, 3.141563, -0.000000]),accel_mss,speed_ms,0,0.001)
      movel(pose_trans(ref_frame,p[0.017507, 0.135155, -0.000125, -0.013708, 3.141563, 0.000000]),accel_mss,speed_ms,0,0.001)
      movel(pose_trans(ref_frame,p[0.017355, 0.135138, -0.000125, -0.013708, 3.141563, 0.000000]),accel_mss,speed_ms,0,0.001)
      movel(pose_trans(ref_frame,p[0.017203, 0.135126, -0.000125, -0.013708, 3.141563, -0.000000]),accel_mss,speed_ms,0,0.001)
      movel(pose_trans(ref_frame,p[0.017034, 0.135118, -0.000125, -0.013708, 3.141563, 0.000000]),accel_mss,speed_ms,0,0.001)
      movel(pose_trans(ref_frame,p[0.016865, 0.135115, -0.000125, -0.013708, 3.141563, -0.000000]),accel_mss,speed_ms,0,0.001)
      movel(pose_trans(ref_frame,p[0.016008, 0.135109, -0.000125, -0.013708, 3.141563, -0.000000]),accel_mss,speed_ms,0,0.001)
      movel(pose_trans(ref_frame,p[0.016011, 0.134006, -0.000125, -0.013708, 3.141563, -0.000000]),accel_mss,speed_ms,0,0) # end trace
      speed_ms    = 1.000
      movel(pose_trans(ref_frame,p[0.016011, 0.134006, 0.005000, -0.013708, 3.141563, -0.000000]),accel_mss,speed_ms,0,0.001)
      movel(pose_trans(ref_frame,p[0.000000, 0.000000, 0.005000, -0.013708, 3.141563, 0.000000]),accel_mss,speed_ms,0,0.001)
      movel(pose_trans(ref_frame,p[0.000000, 0.000000, 0.055000, -0.013708, 3.141563, -0.000000]),accel_mss,speed_ms,0,0.001)
      # End of main program
    end

    output_0028()
    $ 3 "MoveJ"
    $ 4 "Waypoint_1" "breakAfter"
    movej(get_inverse_kin(Waypoint_1_p, qnear=Waypoint_1_q), a=1.3962634015954636, v=1.0471975511965976)
    $ 5 "Halt"
    halt
  end
end
